LIN {X 0.048,Y -476.705,Z 798.727,A 0.000,B 0.000,C 90.000,E1 346.825} C_DIS
LIN {X -0.156,Y -479.692,Z 798.725,A 0.000,B 0.000,C 90.000,E1 346.589} C_DIS
LIN {X 0.040,Y -487.242,Z 798.722,A 0.000,B 0.000,C 90.000,E1 345.992} C_DIS
LIN {X -0.210,Y -497.903,Z 798.718,A 0.000,B 0.000,C 90.000,E1 345.283} C_DIS
LIN {X -0.076,Y -513.435,Z 798.712,A 0.000,B 0.000,C 90.000,E1 344.212} C_DIS
LIN {X -0.131,Y -527.592,Z 798.707,A 0.000,B 0.000,C 90.000,E1 343.268} C_DIS
LIN {X 0.119,Y -536.840,Z 798.703,A 0.000,B 0.000,C 90.000,E1 342.598} C_DIS
LIN {X 0.066,Y -545.875,Z 798.700,A 0.000,B 0.000,C 90.000,E1 341.945} C_DIS
LIN {X -0.103,Y -553.277,Z 798.697,A 0.000,B 0.000,C 90.000,E1 341.402} C_DIS
LIN {X 0.117,Y -561.468,Z 798.693,A 0.000,B 0.000,C 90.000,E1 340.678} C_DIS
LIN {X 0.102,Y -566.684,Z 798.690,A 0.000,B 0.000,C 90.000,E1 340.188} C_DIS
LIN {X -0.162,Y -570.455,Z 798.688,A 0.000,B 0.000,C 90.000,E1 339.826} C_DIS
LIN {X 0.032,Y -575.308,Z 798.685,A 0.000,B 0.000,C 90.000,E1 339.263} C_DIS
LIN {X -0.045,Y -580.753,Z 798.681,A 0.000,B 0.000,C 90.000,E1 338.592} C_DIS
LIN {X -0.081,Y -585.828,Z 798.677,A 0.000,B 0.000,C 90.000,E1 337.922} C_DIS
LIN {X 0.150,Y -590.581,Z 798.674,A 0.000,B 0.000,C 90.000,E1 337.230} C_DIS
LIN {X -0.352,Y -595.110,Z 798.670,A 0.000,B 0.000,C 90.000,E1 336.613} C_DIS
LIN {X -0.151,Y -601.960,Z 798.664,A 0.000,B 0.000,C 90.000,E1 335.537} C_DIS
LIN {X 0.153,Y -608.398,Z 798.658,A 0.000,B 0.000,C 90.000,E1 334.460} C_DIS
LIN {X 0.000,Y -614.526,Z 798.652,A 0.000,B 0.000,C 90.000,E1 333.435} C_DIS
LIN {X -0.063,Y -618.848,Z 798.648,A 0.000,B 0.000,C 90.000,E1 332.666} C_DIS
LIN {X -0.084,Y -623.726,Z 798.643,A 0.000,B 0.000,C 90.000,E1 331.769} C_DIS
LIN {X -0.071,Y -627.030,Z 798.640,A 0.000,B 0.000,C 90.000,E1 331.129} C_DIS
LIN {X -0.208,Y -633.548,Z 798.633,A 0.000,B 0.000,C 90.000,E1 329.871} C_DIS
LIN {X -0.288,Y -638.306,Z 798.627,A 0.000,B 0.000,C 90.000,E1 328.869} C_DIS
LIN {X 0.182,Y -641.636,Z 798.623,A 0.000,B 0.000,C 90.000,E1 328.074} C_DIS
LIN {X -0.345,Y -645.875,Z 798.617,A 0.000,B 0.000,C 90.000,E1 327.120} C_DIS
LIN {X 0.079,Y -649.887,Z 798.612,A 0.000,B 0.000,C 90.000,E1 326.087} C_DIS
LIN {X 0.096,Y -654.439,Z 798.605,A 0.000,B 0.000,C 90.000,E1 324.848} C_DIS
LIN {X 0.095,Y -657.747,Z 798.599,A 0.000,B 0.000,C 90.000,E1 323.863} C_DIS
LIN {X 0.056,Y -660.091,Z 798.595,A 0.000,B 0.000,C 90.000,E1 323.130} C_DIS
LIN {X 0.062,Y -664.567,Z 798.587,A 0.000,B 0.000,C 90.000,E1 321.662} C_DIS
LIN {X 0.166,Y -667.889,Z 798.580,A 0.000,B 0.000,C 90.000,E1 320.436} C_DIS
LIN {X 0.233,Y -670.845,Z 798.574,A 0.000,B 0.000,C 90.000,E1 319.218} C_DIS
LIN {X -0.082,Y -674.221,Z 798.566,A 0.000,B 0.000,C 90.000,E1 317.796} C_DIS
LIN {X -0.039,Y -675.220,Z 798.563,A 0.000,B 0.000,C 90.000,E1 317.310} C_DIS
LIN {X -0.389,Y -677.131,Z 798.557,A 0.000,B 0.000,C 90.000,E1 316.377} C_DIS
LIN {X -0.248,Y -678.801,Z 798.552,A 0.000,B 0.000,C 90.000,E1 315.405} C_DIS
LIN {X -0.037,Y -680.720,Z 798.546,A 0.000,B 0.000,C 90.000,E1 314.190} C_DIS
LIN {X -0.219,Y -682.747,Z 798.538,A 0.000,B 0.000,C 90.000,E1 312.771} C_DIS
LIN {X 0.089,Y -684.304,Z 798.531,A 0.000,B 0.000,C 90.000,E1 311.553} C_DIS
LIN {X -0.147,Y -685.497,Z 798.526,A 0.000,B 0.000,C 90.000,E1 310.620} C_DIS
LIN {X 0.198,Y -686.778,Z 798.519,A 0.000,B 0.000,C 90.000,E1 309.402} C_DIS
LIN {X 0.120,Y -687.963,Z 798.512,A 0.000,B 0.000,C 90.000,E1 308.222} C_DIS
LIN {X 0.232,Y -689.299,Z 798.505,A 0.000,B 0.000,C 90.000,E1 306.790} C_DIS
LIN {X -0.032,Y -690.506,Z 798.497,A 0.000,B 0.000,C 90.000,E1 305.391} C_DIS
LIN {X 0.090,Y -691.413,Z 798.490,A 0.000,B 0.000,C 90.000,E1 304.199} C_DIS
LIN {X 0.084,Y -692.648,Z 798.481,A 0.000,B 0.000,C 90.000,E1 302.546} C_DIS
LIN {X -0.033,Y -694.068,Z 798.470,A 0.000,B 0.000,C 90.000,E1 300.669} C_DIS
LIN {X -0.004,Y -694.849,Z 798.464,A 0.000,B 0.000,C 90.000,E1 299.489} C_DIS
LIN {X -0.063,Y -695.800,Z 798.455,A 0.000,B 0.000,C 90.000,E1 297.847} C_DIS
LIN {X -0.177,Y -696.974,Z 798.444,A 0.000,B 0.000,C 90.000,E1 295.976} C_DIS
LIN {X 0.197,Y -697.824,Z 798.438,A 0.000,B 0.000,C 90.000,E1 294.771} C_DIS
LIN {X -0.204,Y -697.968,Z 798.435,A 0.000,B 0.000,C 90.000,E1 294.335} C_DIS
LIN {X 0.058,Y -697.877,Z 798.434,A 0.000,B 0.000,C 90.000,E1 294.079} C_DIS
LIN {X -0.342,Y -697.307,Z 798.431,A 0.000,B 0.000,C 90.000,E1 293.643} C_DIS
LIN {X -0.083,Y -696.495,Z 798.430,A 0.000,B 0.000,C 90.000,E1 293.387} C_DIS
LIN {X 0.150,Y -693.935,Z 798.427,A 0.000,B 0.000,C 90.000,E1 292.898} C_DIS
LIN {X 0.272,Y -693.079,Z 798.427,A 0.000,B 0.000,C 90.000,E1 292.770} C_DIS
LIN {X 0.394,Y -691.818,Z 798.426,A 0.000,B 0.000,C 90.000,E1 292.642} C_DIS
LIN {X -0.180,Y -687.922,Z 798.425,A 0.000,B 0.000,C 90.000,E1 292.461} C_DIS
LIN {X -0.053,Y -684.888,Z 798.424,A 0.000,B 0.000,C 90.000,E1 292.280} C_DIS
LIN {X -0.186,Y -683.041,Z 798.423,A 0.000,B 0.000,C 90.000,E1 292.206} C_DIS
LIN {X -0.099,Y -674.904,Z 798.422,A 0.000,B 0.000,C 90.000,E1 291.950} C_DIS
LIN {X -0.081,Y -673.076,Z 798.422,A 0.000,B 0.000,C 90.000,E1 291.897} C_DIS
LIN {X 0.152,Y -663.499,Z 798.421,A 0.000,B 0.000,C 90.000,E1 291.716} C_DIS
LIN {X -0.331,Y -649.518,Z 798.420,A 0.000,B 0.000,C 90.000,E1 291.535} C_DIS
LIN {X -0.273,Y -635.379,Z 798.418,A 0.000,B 0.000,C 90.000,E1 291.280} C_DIS
LIN {X -0.207,Y -618.231,Z 798.416,A 0.000,B 0.000,C 90.000,E1 290.918} C_DIS
LIN {X 0.086,Y -605.022,Z 798.414,A 0.000,B 0.000,C 90.000,E1 290.556} C_DIS
LIN {X -0.042,Y -598.409,Z 798.413,A 0.000,B 0.000,C 90.000,E1 290.375} C_DIS
LIN {X -0.004,Y -585.106,Z 798.411,A 0.000,B 0.000,C 90.000,E1 289.939} C_DIS
LIN {X 0.004,Y -574.115,Z 798.408,A 0.000,B 0.000,C 90.000,E1 289.504} C_DIS
LIN {X -0.070,Y -568.690,Z 798.407,A 0.000,B 0.000,C 90.000,E1 289.214} C_DIS
LIN {X -0.174,Y -566.213,Z 798.405,A 0.000,B 0.000,C 90.000,E1 288.960} C_DIS
LIN {X -0.111,Y -565.126,Z 798.405,A 0.000,B 0.000,C 90.000,E1 288.852} C_DIS
LIN {X -0.016,Y -564.192,Z 798.404,A 0.000,B 0.000,C 90.000,E1 288.671} C_DIS
LIN {X -0.119,Y -563.612,Z 798.403,A 0.000,B 0.000,C 90.000,E1 288.544} C_DIS
LIN {X 0.123,Y -563.320,Z 798.402,A 0.000,B 0.000,C 90.000,E1 288.362} C_DIS
LIN {X -0.095,Y -562.507,Z 798.401,A 0.000,B 0.000,C 90.000,E1 288.109} C_DIS
LIN {X 0.045,Y -562.296,Z 798.399,A 0.000,B 0.000,C 90.000,E1 287.819} C_DIS
LIN {X 0.186,Y -562.165,Z 798.398,A 0.000,B 0.000,C 90.000,E1 287.528} C_DIS
LIN {X 0.073,Y -562.226,Z 798.397,A 0.000,B 0.000,C 90.000,E1 287.402} C_DIS
LIN {X -0.127,Y -564.221,Z 798.393,A 0.000,B 0.000,C 90.000,E1 286.732} C_DIS
LIN {X 0.136,Y -565.076,Z 798.392,A 0.000,B 0.000,C 90.000,E1 286.567} C_DIS
LIN {X 0.180,Y -568.381,Z 798.390,A 0.000,B 0.000,C 90.000,E1 286.150} C_DIS
LIN {X 0.070,Y -569.256,Z 798.389,A 0.000,B 0.000,C 90.000,E1 286.024} C_DIS
LIN {X -0.235,Y -572.706,Z 798.385,A 0.000,B 0.000,C 90.000,E1 285.371} C_DIS
LIN {X 0.103,Y -573.656,Z 798.384,A 0.000,B 0.000,C 90.000,E1 285.064} C_DIS
LIN {X -0.220,Y -576.381,Z 798.378,A 0.000,B 0.000,C 90.000,E1 284.008} C_DIS
LIN {X -0.013,Y -576.591,Z 798.376,A 0.000,B 0.000,C 90.000,E1 283.716} C_DIS
LIN {X -0.020,Y -576.495,Z 798.373,A 0.000,B 0.000,C 90.000,E1 283.175} C_DIS
LIN {X 0.190,Y -576.235,Z 798.372,A 0.000,B 0.000,C 90.000,E1 282.883} C_DIS
LIN {X -0.161,Y -575.837,Z 798.370,A 0.000,B 0.000,C 90.000,E1 282.647} C_DIS
LIN {X 0.256,Y -573.735,Z 798.367,A 0.000,B 0.000,C 90.000,E1 282.063} C_DIS
LIN {X -0.100,Y -572.413,Z 798.366,A 0.000,B 0.000,C 90.000,E1 281.827} C_DIS
LIN {X -0.143,Y -569.026,Z 798.363,A 0.000,B 0.000,C 90.000,E1 281.422} C_DIS
LIN {X 0.123,Y -566.344,Z 798.362,A 0.000,B 0.000,C 90.000,E1 281.130} C_DIS
LIN {X 0.232,Y -562.560,Z 798.361,A 0.000,B 0.000,C 90.000,E1 280.894} C_DIS
LIN {X -0.156,Y -560.238,Z 798.360,A 0.000,B 0.000,C 90.000,E1 280.838} C_DIS
LIN {X -0.294,Y -558.014,Z 798.360,A 0.000,B 0.000,C 90.000,E1 280.782} C_DIS
LIN {X 0.219,Y -556.305,Z 798.359,A 0.000,B 0.000,C 90.000,E1 280.658} C_DIS
LIN {X -0.099,Y -555.281,Z 798.359,A 0.000,B 0.000,C 90.000,E1 280.602} C_DIS
LIN {X -0.134,Y -552.696,Z 798.357,A 0.000,B 0.000,C 90.000,E1 280.310} C_DIS
LIN {X 0.133,Y -552.209,Z 798.357,A 0.000,B 0.000,C 90.000,E1 280.197} C_DIS
LIN {X 0.017,Y -551.503,Z 798.354,A 0.000,B 0.000,C 90.000,E1 279.792} C_DIS
LIN {X 0.215,Y -550.863,Z 798.342,A 0.000,B 0.000,C 90.000,E1 277.530} C_DIS
LIN {X 0.166,Y -550.166,Z 798.333,A 0.000,B 0.000,C 90.000,E1 275.853} C_DIS
LIN {X -0.105,Y -549.616,Z 798.326,A 0.000,B 0.000,C 90.000,E1 274.759} C_DIS
LIN {X 0.122,Y -548.967,Z 798.320,A 0.000,B 0.000,C 90.000,E1 273.612} C_DIS
LIN {X -0.108,Y -547.797,Z 798.311,A 0.000,B 0.000,C 90.000,E1 271.949} C_DIS
LIN {X 0.140,Y -546.886,Z 798.303,A 0.000,B 0.000,C 90.000,E1 270.516} C_DIS
LIN {X -0.187,Y -545.959,Z 798.295,A 0.000,B 0.000,C 90.000,E1 269.141} C_DIS
LIN {X 0.097,Y -544.570,Z 798.284,A 0.000,B 0.000,C 90.000,E1 267.135} C_DIS
LIN {X -0.201,Y -543.491,Z 798.275,A 0.000,B 0.000,C 90.000,E1 265.469} C_DIS
LIN {X -0.003,Y -542.620,Z 798.267,A 0.000,B 0.000,C 90.000,E1 264.033} C_DIS
LIN {X 0.229,Y -541.566,Z 798.259,A 0.000,B 0.000,C 90.000,E1 262.591} C_DIS
LIN {X 0.059,Y -540.107,Z 798.250,A 0.000,B 0.000,C 90.000,E1 260.905} C_DIS
LIN {X 0.257,Y -539.053,Z 798.243,A 0.000,B 0.000,C 90.000,E1 259.746} C_DIS
LIN {X 0.139,Y -537.415,Z 798.234,A 0.000,B 0.000,C 90.000,E1 258.049} C_DIS
LIN {X -0.019,Y -535.728,Z 798.224,A 0.000,B 0.000,C 90.000,E1 256.353} C_DIS
LIN {X -0.147,Y -534.186,Z 798.216,A 0.000,B 0.000,C 90.000,E1 254.936} C_DIS
LIN {X 0.022,Y -532.181,Z 798.207,A 0.000,B 0.000,C 90.000,E1 253.196} C_DIS
LIN {X -0.030,Y -530.495,Z 798.199,A 0.000,B 0.000,C 90.000,E1 251.764} C_DIS
LIN {X 0.041,Y -528.664,Z 798.191,A 0.000,B 0.000,C 90.000,E1 250.315} C_DIS
LIN {X 0.078,Y -527.108,Z 798.184,A 0.000,B 0.000,C 90.000,E1 249.156} C_DIS
LIN {X 0.139,Y -524.559,Z 798.175,A 0.000,B 0.000,C 90.000,E1 247.411} C_DIS
LIN {X 0.153,Y -521.953,Z 798.165,A 0.000,B 0.000,C 90.000,E1 245.665} C_DIS
LIN {X 0.178,Y -519.658,Z 798.157,A 0.000,B 0.000,C 90.000,E1 244.204} C_DIS
LIN {X 0.157,Y -517.176,Z 798.149,A 0.000,B 0.000,C 90.000,E1 242.743} C_DIS
LIN {X -0.133,Y -514.636,Z 798.141,A 0.000,B 0.000,C 90.000,E1 241.307} C_DIS
LIN {X 0.230,Y -511.862,Z 798.132,A 0.000,B 0.000,C 90.000,E1 239.793} C_DIS
LIN {X -0.238,Y -509.540,Z 798.126,A 0.000,B 0.000,C 90.000,E1 238.663} C_DIS
LIN {X -0.145,Y -506.520,Z 798.118,A 0.000,B 0.000,C 90.000,E1 237.168} C_DIS
LIN {X -0.004,Y -503.984,Z 798.111,A 0.000,B 0.000,C 90.000,E1 235.960} C_DIS
LIN {X -0.277,Y -499.922,Z 798.101,A 0.000,B 0.000,C 90.000,E1 234.196} C_DIS
LIN {X 0.189,Y -496.161,Z 798.093,A 0.000,B 0.000,C 90.000,E1 232.637} C_DIS
LIN {X -0.042,Y -491.609,Z 798.083,A 0.000,B 0.000,C 90.000,E1 230.848} C_DIS
LIN {X 0.130,Y -485.202,Z 798.067,A 0.000,B 0.000,C 90.000,E1 228.081} C_DIS
LIN {X -0.249,Y -480.588,Z 798.055,A 0.000,B 0.000,C 90.000,E1 225.972} C_DIS
LIN {X -0.195,Y -476.476,Z 798.045,A 0.000,B 0.000,C 90.000,E1 224.109} C_DIS
LIN {X -0.127,Y -471.709,Z 798.033,A 0.000,B 0.000,C 90.000,E1 221.919} C_DIS
LIN {X 0.088,Y -467.690,Z 798.022,A 0.000,B 0.000,C 90.000,E1 220.011} C_DIS
LIN {X -0.146,Y -464.455,Z 798.014,A 0.000,B 0.000,C 90.000,E1 218.463} C_DIS
LIN {X 0.059,Y -459.854,Z 798.001,A 0.000,B 0.000,C 90.000,E1 216.217} C_DIS
LIN {X -0.136,Y -455.828,Z 797.991,A 0.000,B 0.000,C 90.000,E1 214.326} C_DIS
LIN {X 0.038,Y -451.298,Z 797.978,A 0.000,B 0.000,C 90.000,E1 212.054} C_DIS
LIN {X -0.082,Y -447.415,Z 797.967,A 0.000,B 0.000,C 90.000,E1 210.129} C_DIS
LIN {X 0.097,Y -443.579,Z 797.957,A 0.000,B 0.000,C 90.000,E1 208.153} C_DIS
LIN {X -0.070,Y -440.543,Z 797.947,A 0.000,B 0.000,C 90.000,E1 206.539} C_DIS
LIN {X 0.155,Y -436.121,Z 797.935,A 0.000,B 0.000,C 90.000,E1 204.207} C_DIS
LIN {X -0.125,Y -432.889,Z 797.925,A 0.000,B 0.000,C 90.000,E1 202.589} C_DIS
LIN {X -0.067,Y -429.687,Z 797.916,A 0.000,B 0.000,C 90.000,E1 200.918} C_DIS
LIN {X 0.170,Y -425.220,Z 797.903,A 0.000,B 0.000,C 90.000,E1 198.544} C_DIS
LIN {X -0.001,Y -422.607,Z 797.896,A 0.000,B 0.000,C 90.000,E1 197.221} C_DIS
LIN {X -0.160,Y -419.352,Z 797.886,A 0.000,B 0.000,C 90.000,E1 195.552} C_DIS
LIN {X 0.210,Y -414.775,Z 797.873,A 0.000,B 0.000,C 90.000,E1 193.119} C_DIS
LIN {X 0.023,Y -412.875,Z 797.867,A 0.000,B 0.000,C 90.000,E1 192.119} C_DIS
LIN {X -0.075,Y -408.571,Z 797.854,A 0.000,B 0.000,C 90.000,E1 189.726} C_DIS
LIN {X -0.059,Y -406.165,Z 797.846,A 0.000,B 0.000,C 90.000,E1 188.341} C_DIS
LIN {X -0.021,Y -403.637,Z 797.839,A 0.000,B 0.000,C 90.000,E1 186.947} C_DIS
LIN {X -0.135,Y -400.464,Z 797.829,A 0.000,B 0.000,C 90.000,E1 185.220} C_DIS
LIN {X -0.017,Y -393.717,Z 797.804,A 0.000,B 0.000,C 90.000,E1 180.630} C_DIS
LIN {X 0.090,Y -390.124,Z 797.786,A 0.000,B 0.000,C 90.000,E1 177.421} C_DIS
LIN {X -0.025,Y -387.841,Z 797.774,A 0.000,B 0.000,C 90.000,E1 175.298} C_DIS
LIN {X -0.132,Y -385.637,Z 797.762,A 0.000,B 0.000,C 90.000,E1 173.166} C_DIS
LIN {X 0.135,Y -383.530,Z 797.750,A 0.000,B 0.000,C 90.000,E1 170.971} C_DIS
LIN {X -0.083,Y -381.070,Z 797.734,A 0.000,B 0.000,C 90.000,E1 168.117} C_DIS
LIN {X -0.140,Y -378.783,Z 797.716,A 0.000,B 0.000,C 90.000,E1 164.866} C_DIS
LIN {X -0.097,Y -376.970,Z 797.694,A 0.000,B 0.000,C 90.000,E1 160.859} C_DIS
LIN {X 0.037,Y -377.905,Z 797.649,A 0.000,B 0.000,C 90.000,E1 152.820} C_DIS
LIN {X 0.180,Y -380.213,Z 797.635,A 0.000,B 0.000,C 90.000,E1 150.255} C_DIS
LIN {X -0.052,Y -381.817,Z 797.629,A 0.000,B 0.000,C 90.000,E1 149.203} C_DIS
LIN {X 0.077,Y -384.673,Z 797.621,A 0.000,B 0.000,C 90.000,E1 147.740} C_DIS
LIN {X 0.136,Y -388.637,Z 797.613,A 0.000,B 0.000,C 90.000,E1 146.294} C_DIS
LIN {X -0.125,Y -392.389,Z 797.607,A 0.000,B 0.000,C 90.000,E1 145.261} C_DIS
LIN {X 0.107,Y -394.977,Z 797.604,A 0.000,B 0.000,C 90.000,E1 144.609} C_DIS
LIN {X 0.058,Y -398.597,Z 797.600,A 0.000,B 0.000,C 90.000,E1 143.909} C_DIS
LIN {X 0.009,Y -402.309,Z 797.596,A 0.000,B 0.000,C 90.000,E1 143.290} C_DIS
LIN {X 0.188,Y -407.473,Z 797.592,A 0.000,B 0.000,C 90.000,E1 142.477} C_DIS
LIN {X 0.122,Y -416.188,Z 797.585,A 0.000,B 0.000,C 90.000,E1 141.331} C_DIS
LIN {X -0.063,Y -425.883,Z 797.579,A 0.000,B 0.000,C 90.000,E1 140.194} C_DIS
LIN {X 0.075,Y -433.645,Z 797.573,A 0.000,B 0.000,C 90.000,E1 139.175} C_DIS
LIN {X 0.162,Y -446.410,Z 797.564,A 0.000,B 0.000,C 90.000,E1 137.553} C_DIS
LIN {X 0.166,Y -451.691,Z 797.561,A 0.000,B 0.000,C 90.000,E1 136.905} C_DIS
LIN {X 0.078,Y -459.089,Z 797.555,A 0.000,B 0.000,C 90.000,E1 135.972} C_DIS
LIN {X -0.001,Y -463.712,Z 797.552,A 0.000,B 0.000,C 90.000,E1 135.364} C_DIS
LIN {X 0.007,Y -473.709,Z 797.544,A 0.000,B 0.000,C 90.000,E1 133.947} C_DIS
LIN {X 0.141,Y -480.131,Z 797.539,A 0.000,B 0.000,C 90.000,E1 133.014} C_DIS
LIN {X 0.268,Y -487.242,Z 797.533,A 0.000,B 0.000,C 90.000,E1 131.919} C_DIS
LIN {X 0.248,Y -495.005,Z 797.526,A 0.000,B 0.000,C 90.000,E1 130.701} C_DIS
LIN {X 0.117,Y -502.992,Z 797.519,A 0.000,B 0.000,C 90.000,E1 129.358} C_DIS
LIN {X -0.004,Y -507.287,Z 797.515,A 0.000,B 0.000,C 90.000,E1 128.624} C_DIS
LIN {X -0.059,Y -513.696,Z 797.508,A 0.000,B 0.000,C 90.000,E1 127.443} C_DIS
LIN {X -0.279,Y -518.187,Z 797.503,A 0.000,B 0.000,C 90.000,E1 126.583} C_DIS
LIN {X -0.028,Y -522.549,Z 797.498,A 0.000,B 0.000,C 90.000,E1 125.678} C_DIS
LIN {X -0.024,Y -527.143,Z 797.493,A 0.000,B 0.000,C 90.000,E1 124.692} C_DIS
LIN {X 0.002,Y -533.141,Z 797.485,A 0.000,B 0.000,C 90.000,E1 123.245} C_DIS
LIN {X -0.322,Y -536.545,Z 797.480,A 0.000,B 0.000,C 90.000,E1 122.418} C_DIS
LIN {X -0.157,Y -540.829,Z 797.474,A 0.000,B 0.000,C 90.000,E1 121.258} C_DIS
LIN {X 0.051,Y -543.851,Z 797.469,A 0.000,B 0.000,C 90.000,E1 120.384} C_DIS
LIN {X -0.232,Y -547.520,Z 797.463,A 0.000,B 0.000,C 90.000,E1 119.283} C_DIS
LIN {X 0.055,Y -551.711,Z 797.455,A 0.000,B 0.000,C 90.000,E1 117.847} C_DIS
LIN {X -0.152,Y -553.269,Z 797.452,A 0.000,B 0.000,C 90.000,E1 117.308} C_DIS
LIN {X 0.163,Y -555.267,Z 797.447,A 0.000,B 0.000,C 90.000,E1 116.437} C_DIS
LIN {X 0.039,Y -557.302,Z 797.441,A 0.000,B 0.000,C 90.000,E1 115.335} C_DIS
LIN {X 0.118,Y -558.260,Z 797.438,A 0.000,B 0.000,C 90.000,E1 114.771} C_DIS
LIN {X -0.213,Y -559.661,Z 797.432,A 0.000,B 0.000,C 90.000,E1 113.695} C_DIS
LIN {X -0.235,Y -560.865,Z 797.425,A 0.000,B 0.000,C 90.000,E1 112.589} C_DIS
LIN {X 0.088,Y -562.248,Z 797.418,A 0.000,B 0.000,C 90.000,E1 111.173} C_DIS
LIN {X -0.097,Y -563.346,Z 797.410,A 0.000,B 0.000,C 90.000,E1 109.812} C_DIS
LIN {X 0.065,Y -564.073,Z 797.402,A 0.000,B 0.000,C 90.000,E1 108.417} C_DIS
LIN {X -0.321,Y -564.895,Z 797.393,A 0.000,B 0.000,C 90.000,E1 106.804} C_DIS
LIN {X 0.170,Y -565.967,Z 797.383,A 0.000,B 0.000,C 90.000,E1 104.828} C_DIS
LIN {X -0.161,Y -567.198,Z 797.372,A 0.000,B 0.000,C 90.000,E1 102.939} C_DIS
LIN {X 0.164,Y -568.222,Z 797.364,A 0.000,B 0.000,C 90.000,E1 101.535} C_DIS
LIN {X -0.156,Y -569.282,Z 797.357,A 0.000,B 0.000,C 90.000,E1 100.197} C_DIS
LIN {X 0.109,Y -570.390,Z 797.349,A 0.000,B 0.000,C 90.000,E1 98.803} C_DIS
LIN {X -0.069,Y -571.516,Z 797.340,A 0.000,B 0.000,C 90.000,E1 97.182} C_DIS
LIN {X -0.034,Y -572.182,Z 797.334,A 0.000,B 0.000,C 90.000,E1 96.087} C_DIS
LIN {X -0.115,Y -573.264,Z 797.323,A 0.000,B 0.000,C 90.000,E1 94.188} C_DIS
LIN {X -0.067,Y -573.781,Z 797.317,A 0.000,B 0.000,C 90.000,E1 93.094} C_DIS
LIN {X 0.235,Y -574.510,Z 797.308,A 0.000,B 0.000,C 90.000,E1 91.432} C_DIS
LIN {X -0.180,Y -574.948,Z 797.301,A 0.000,B 0.000,C 90.000,E1 90.115} C_DIS
LIN {X 0.139,Y -575.545,Z 797.292,A 0.000,B 0.000,C 90.000,E1 88.453} C_DIS
LIN {X -0.068,Y -575.967,Z 797.282,A 0.000,B 0.000,C 90.000,E1 86.846} C_DIS
LIN {X -0.107,Y -576.439,Z 797.272,A 0.000,B 0.000,C 90.000,E1 84.951} C_DIS
LIN {X 0.136,Y -576.695,Z 797.264,A 0.000,B 0.000,C 90.000,E1 83.571} C_DIS
LIN {X 0.079,Y -576.993,Z 797.255,A 0.000,B 0.000,C 90.000,E1 81.951} C_DIS
LIN {X 0.029,Y -577.292,Z 797.246,A 0.000,B 0.000,C 90.000,E1 80.330} C_DIS
LIN {X -0.141,Y -577.537,Z 797.239,A 0.000,B 0.000,C 90.000,E1 78.993} C_DIS
LIN {X -0.197,Y -577.585,Z 797.231,A 0.000,B 0.000,C 90.000,E1 77.645} C_DIS
LIN {X 0.099,Y -577.526,Z 797.222,A 0.000,B 0.000,C 90.000,E1 75.992} C_DIS
LIN {X 0.184,Y -577.316,Z 797.215,A 0.000,B 0.000,C 90.000,E1 74.629} C_DIS
LIN {X 0.073,Y -577.068,Z 797.206,A 0.000,B 0.000,C 90.000,E1 73.015} C_DIS
LIN {X 0.306,Y -576.761,Z 797.198,A 0.000,B 0.000,C 90.000,E1 71.638} C_DIS
LIN {X -0.207,Y -576.390,Z 797.192,A 0.000,B 0.000,C 90.000,E1 70.604} C_DIS
LIN {X 0.189,Y -575.896,Z 797.185,A 0.000,B 0.000,C 90.000,E1 69.209} C_DIS
LIN {X -0.133,Y -575.419,Z 797.179,A 0.000,B 0.000,C 90.000,E1 68.156} C_DIS
LIN {X -0.088,Y -574.714,Z 797.171,A 0.000,B 0.000,C 90.000,E1 66.794} C_DIS
LIN {X 0.331,Y -574.047,Z 797.165,A 0.000,B 0.000,C 90.000,E1 65.665} C_DIS
LIN {X 0.218,Y -573.334,Z 797.159,A 0.000,B 0.000,C 90.000,E1 64.588} C_DIS
LIN {X 0.095,Y -572.520,Z 797.153,A 0.000,B 0.000,C 90.000,E1 63.512} C_DIS
LIN {X 0.216,Y -571.490,Z 797.147,A 0.000,B 0.000,C 90.000,E1 62.410} C_DIS
LIN {X -0.283,Y -570.602,Z 797.142,A 0.000,B 0.000,C 90.000,E1 61.641} C_DIS
LIN {X -0.194,Y -569.232,Z 797.136,A 0.000,B 0.000,C 90.000,E1 60.539} C_DIS
LIN {X 0.152,Y -567.652,Z 797.130,A 0.000,B 0.000,C 90.000,E1 59.410} C_DIS
LIN {X -0.114,Y -566.325,Z 797.126,A 0.000,B 0.000,C 90.000,E1 58.614} C_DIS
LIN {X -0.097,Y -564.856,Z 797.121,A 0.000,B 0.000,C 90.000,E1 57.788} C_DIS
LIN {X -0.089,Y -563.185,Z 797.116,A 0.000,B 0.000,C 90.000,E1 56.962} C_DIS
LIN {X -0.313,Y -560.700,Z 797.110,A 0.000,B 0.000,C 90.000,E1 55.881} C_DIS
LIN {X -0.264,Y -557.786,Z 797.104,A 0.000,B 0.000,C 90.000,E1 54.769} C_DIS
LIN {X -0.011,Y -555.414,Z 797.100,A 0.000,B 0.000,C 90.000,E1 53.909} C_DIS
LIN {X 0.145,Y -553.662,Z 797.096,A 0.000,B 0.000,C 90.000,E1 53.336} C_DIS
LIN {X 0.353,Y -550.803,Z 797.092,A 0.000,B 0.000,C 90.000,E1 52.477} C_DIS
LIN {X -0.298,Y -548.790,Z 797.089,A 0.000,B 0.000,C 90.000,E1 51.984} C_DIS
LIN {X 0.193,Y -545.353,Z 797.084,A 0.000,B 0.000,C 90.000,E1 51.090} C_DIS
LIN {X -0.149,Y -542.914,Z 797.081,A 0.000,B 0.000,C 90.000,E1 50.561} C_DIS
LIN {X -0.094,Y -540.266,Z 797.078,A 0.000,B 0.000,C 90.000,E1 49.989} C_DIS
LIN {X -0.291,Y -534.898,Z 797.072,A 0.000,B 0.000,C 90.000,E1 49.013} C_DIS
LIN {X 0.057,Y -533.336,Z 797.071,A 0.000,B 0.000,C 90.000,E1 48.690} C_DIS
LIN {X -0.200,Y -528.678,Z 797.067,A 0.000,B 0.000,C 90.000,E1 48.000} C_DIS
LIN {X 0.089,Y -524.643,Z 797.063,A 0.000,B 0.000,C 90.000,E1 47.391} C_DIS
LIN {X -0.189,Y -521.357,Z 797.061,A 0.000,B 0.000,C 90.000,E1 46.986} C_DIS
LIN {X 0.040,Y -516.511,Z 797.058,A 0.000,B 0.000,C 90.000,E1 46.377} C_DIS
LIN {X 0.111,Y -507.647,Z 797.052,A 0.000,B 0.000,C 90.000,E1 45.405} C_DIS
LIN {X -0.261,Y -500.374,Z 797.049,A 0.000,B 0.000,C 90.000,E1 44.757} C_DIS
LIN {X -0.219,Y -495.926,Z 797.046,A 0.000,B 0.000,C 90.000,E1 44.352} C_DIS
LIN {X 0.293,Y -489.920,Z 797.044,A 0.000,B 0.000,C 90.000,E1 43.785} C_DIS
LIN {X -0.062,Y -482.139,Z 797.040,A 0.000,B 0.000,C 90.000,E1 43.218} C_DIS
LIN {X 0.189,Y -474.147,Z 797.037,A 0.000,B 0.000,C 90.000,E1 42.609} C_DIS
LIN {X -0.018,Y -464.550,Z 797.033,A 0.000,B 0.000,C 90.000,E1 41.962} C_DIS
LIN {X -0.073,Y -446.893,Z 797.026,A 0.000,B 0.000,C 90.000,E1 40.744} C_DIS
LIN {X -0.233,Y -421.708,Z 797.016,A 0.000,B 0.000,C 90.000,E1 38.910} C_DIS
LIN {X 0.056,Y -407.950,Z 797.010,A 0.000,B 0.000,C 90.000,E1 37.729} C_DIS
LIN {X 0.071,Y -403.546,Z 797.007,A 0.000,B 0.000,C 90.000,E1 37.282} C_DIS
LIN {X 0.028,Y -403.146,Z 797.007,A 0.000,B 0.000,C 90.000,E1 37.237} C_DIS
LIN {X -0.001,Y -403.124,Z 797.007,A 0.000,B 0.000,C 90.000,E1 37.237} C_DIS
LIN {X 0.126,Y -395.009,Z 796.982,A 0.000,B 0.000,C 90.000,E1 32.673} C_DIS
LIN {X -0.212,Y -394.922,Z 796.981,A 0.000,B 0.000,C 90.000,E1 32.546} C_DIS
LIN {X -0.152,Y -395.864,Z 796.966,A 0.000,B 0.000,C 90.000,E1 29.873} C_DIS
LIN {X 0.205,Y -397.336,Z 796.950,A 0.000,B 0.000,C 90.000,E1 27.001} C_DIS
LIN {X 0.140,Y -398.604,Z 796.938,A 0.000,B 0.000,C 90.000,E1 24.899} C_DIS
LIN {X -0.053,Y -400.889,Z 796.921,A 0.000,B 0.000,C 90.000,E1 21.770} C_DIS
LIN {X 0.236,Y -404.220,Z 796.902,A 0.000,B 0.000,C 90.000,E1 18.236} C_DIS
LIN {X -0.208,Y -409.195,Z 796.880,A 0.000,B 0.000,C 90.000,E1 14.481} C_DIS
LIN {X -0.128,Y -413.616,Z 796.865,A 0.000,B 0.000,C 90.000,E1 11.715} C_DIS
LIN {X -0.189,Y -417.166,Z 796.854,A 0.000,B 0.000,C 90.000,E1 9.670} C_DIS
LIN {X 0.044,Y -420.183,Z 796.844,A 0.000,B 0.000,C 90.000,E1 7.936} C_DIS
LIN {X -0.001,Y -423.832,Z 796.833,A 0.000,B 0.000,C 90.000,E1 5.910} C_DIS
LIN {X -0.056,Y -427.559,Z 796.822,A 0.000,B 0.000,C 90.000,E1 3.898} C_DIS
LIN {X -0.069,Y -431.408,Z 796.810,A 0.000,B 0.000,C 90.000,E1 1.892} C_DIS
LIN {X 0.165,Y -435.686,Z 796.799,A 0.000,B 0.000,C 90.000,E1 359.771} C_DIS
LIN {X 0.142,Y -441.483,Z 796.784,A 0.000,B 0.000,C 90.000,E1 357.135} C_DIS
LIN {X 0.208,Y -446.922,Z 796.771,A 0.000,B 0.000,C 90.000,E1 354.837} C_DIS
LIN {X 0.130,Y -450.859,Z 796.763,A 0.000,B 0.000,C 90.000,E1 353.223} C_DIS
LIN {X 0.186,Y -454.754,Z 796.754,A 0.000,B 0.000,C 90.000,E1 351.602} C_DIS
LIN {X -0.126,Y -460.338,Z 796.741,A 0.000,B 0.000,C 90.000,E1 349.398} C_DIS
LIN {X 0.065,Y -462.950,Z 796.737,A 0.000,B 0.000,C 90.000,E1 348.578} C_DIS
LIN {X -0.142,Y -464.261,Z 796.735,A 0.000,B 0.000,C 90.000,E1 348.285} C_DIS
LIN {X 0.112,Y -465.806,Z 796.733,A 0.000,B 0.000,C 90.000,E1 347.937} C_DIS
LIN {X -0.045,Y -468.262,Z 796.731,A 0.000,B 0.000,C 90.000,E1 347.589} C_DIS
LIN {X 0.002,Y -473.215,Z 796.728,A 0.000,B 0.000,C 90.000,E1 346.992} C_DIS
LIN {X -0.049,Y -481.413,Z 796.724,A 0.000,B 0.000,C 90.000,E1 346.284} C_DIS
LIN {X 0.163,Y -490.454,Z 796.720,A 0.000,B 0.000,C 90.000,E1 345.589} C_DIS
LIN {X -0.228,Y -509.270,Z 796.713,A 0.000,B 0.000,C 90.000,E1 344.338} C_DIS
LIN {X 0.045,Y -526.667,Z 796.706,A 0.000,B 0.000,C 90.000,E1 343.142} C_DIS
LIN {X 0.198,Y -535.950,Z 796.703,A 0.000,B 0.000,C 90.000,E1 342.489} C_DIS
LIN {X -0.208,Y -546.506,Z 796.699,A 0.000,B 0.000,C 90.000,E1 341.764} C_DIS
LIN {X 0.242,Y -552.410,Z 796.696,A 0.000,B 0.000,C 90.000,E1 341.275} C_DIS
LIN {X -0.079,Y -560.796,Z 796.692,A 0.000,B 0.000,C 90.000,E1 340.604} C_DIS
LIN {X -0.156,Y -566.114,Z 796.690,A 0.000,B 0.000,C 90.000,E1 340.115} C_DIS
LIN {X 0.061,Y -571.128,Z 796.687,A 0.000,B 0.000,C 90.000,E1 339.571} C_DIS
LIN {X 0.107,Y -575.854,Z 796.684,A 0.000,B 0.000,C 90.000,E1 339.028} C_DIS
LIN {X -0.044,Y -582.271,Z 796.679,A 0.000,B 0.000,C 90.000,E1 338.230} C_DIS
LIN {X 0.090,Y -588.207,Z 796.675,A 0.000,B 0.000,C 90.000,E1 337.411} C_DIS
LIN {X 0.013,Y -594.698,Z 796.669,A 0.000,B 0.000,C 90.000,E1 336.485} C_DIS
LIN {X 0.214,Y -601.571,Z 796.664,A 0.000,B 0.000,C 90.000,E1 335.409} C_DIS
LIN {X -0.294,Y -608.046,Z 796.658,A 0.000,B 0.000,C 90.000,E1 334.409} C_DIS
LIN {X 0.071,Y -614.941,Z 796.651,A 0.000,B 0.000,C 90.000,E1 333.204} C_DIS
LIN {X 0.015,Y -618.553,Z 796.648,A 0.000,B 0.000,C 90.000,E1 332.564} C_DIS
LIN {X 0.277,Y -624.182,Z 796.642,A 0.000,B 0.000,C 90.000,E1 331.513} C_DIS
LIN {X 0.088,Y -630.106,Z 796.636,A 0.000,B 0.000,C 90.000,E1 330.383} C_DIS
LIN {X 0.151,Y -633.403,Z 796.632,A 0.000,B 0.000,C 90.000,E1 329.744} C_DIS
LIN {X 0.092,Y -638.739,Z 796.626,A 0.000,B 0.000,C 90.000,E1 328.614} C_DIS
LIN {X 0.070,Y -643.127,Z 796.620,A 0.000,B 0.000,C 90.000,E1 327.612} C_DIS
LIN {X 0.393,Y -646.307,Z 796.616,A 0.000,B 0.000,C 90.000,E1 326.834} C_DIS
LIN {X -0.139,Y -649.326,Z 796.612,A 0.000,B 0.000,C 90.000,E1 326.135} C_DIS
LIN {X -0.125,Y -653.966,Z 796.605,A 0.000,B 0.000,C 90.000,E1 324.895} C_DIS
LIN {X -0.125,Y -657.346,Z 796.599,A 0.000,B 0.000,C 90.000,E1 323.909} C_DIS
LIN {X 0.363,Y -659.724,Z 796.595,A 0.000,B 0.000,C 90.000,E1 323.130} C_DIS
LIN {X 0.394,Y -663.496,Z 796.589,A 0.000,B 0.000,C 90.000,E1 321.904} C_DIS
LIN {X 0.419,Y -665.599,Z 796.585,A 0.000,B 0.000,C 90.000,E1 321.170} C_DIS
LIN {X -0.049,Y -667.649,Z 796.580,A 0.000,B 0.000,C 90.000,E1 320.481} C_DIS
LIN {X 0.091,Y -670.689,Z 796.574,A 0.000,B 0.000,C 90.000,E1 319.256} C_DIS
LIN {X -0.304,Y -673.576,Z 796.567,A 0.000,B 0.000,C 90.000,E1 318.081} C_DIS
LIN {X 0.234,Y -674.718,Z 796.564,A 0.000,B 0.000,C 90.000,E1 317.553} C_DIS
LIN {X -0.093,Y -677.132,Z 796.558,A 0.000,B 0.000,C 90.000,E1 316.377} C_DIS
LIN {X 0.049,Y -678.799,Z 796.552,A 0.000,B 0.000,C 90.000,E1 315.405} C_DIS
LIN {X 0.261,Y -680.787,Z 796.546,A 0.000,B 0.000,C 90.000,E1 314.190} C_DIS
LIN {X 0.082,Y -682.855,Z 796.538,A 0.000,B 0.000,C 90.000,E1 312.771} C_DIS
LIN {X -0.120,Y -684.435,Z 796.531,A 0.000,B 0.000,C 90.000,E1 311.595} C_DIS
LIN {X 0.104,Y -685.376,Z 796.527,A 0.000,B 0.000,C 90.000,E1 310.862} C_DIS
LIN {X -0.075,Y -686.693,Z 796.521,A 0.000,B 0.000,C 90.000,E1 309.688} C_DIS
LIN {X 0.005,Y -688.135,Z 796.513,A 0.000,B 0.000,C 90.000,E1 308.257} C_DIS
LIN {X -0.418,Y -689.476,Z 796.505,A 0.000,B 0.000,C 90.000,E1 306.870} C_DIS
LIN {X 0.088,Y -690.524,Z 796.498,A 0.000,B 0.000,C 90.000,E1 305.644} C_DIS
LIN {X -0.190,Y -691.431,Z 796.492,A 0.000,B 0.000,C 90.000,E1 304.485} C_DIS
LIN {X 0.411,Y -692.849,Z 796.481,A 0.000,B 0.000,C 90.000,E1 302.546} C_DIS
LIN {X -0.055,Y -694.450,Z 796.469,A 0.000,B 0.000,C 90.000,E1 300.463} C_DIS
LIN {X -0.023,Y -695.181,Z 796.463,A 0.000,B 0.000,C 90.000,E1 299.283} C_DIS
LIN {X -0.082,Y -696.112,Z 796.454,A 0.000,B 0.000,C 90.000,E1 297.641} C_DIS
LIN {X -0.199,Y -697.264,Z 796.443,A 0.000,B 0.000,C 90.000,E1 295.771} C_DIS
LIN {X -0.088,Y -697.928,Z 796.438,A 0.000,B 0.000,C 90.000,E1 294.823} C_DIS
LIN {X 0.145,Y -698.095,Z 796.435,A 0.000,B 0.000,C 90.000,E1 294.335} C_DIS
LIN {X -0.230,Y -698.058,Z 796.434,A 0.000,B 0.000,C 90.000,E1 294.131} C_DIS
LIN {X 0.008,Y -697.411,Z 796.431,A 0.000,B 0.000,C 90.000,E1 293.643} C_DIS
LIN {X 0.266,Y -696.715,Z 796.430,A 0.000,B 0.000,C 90.000,E1 293.387} C_DIS
LIN {X -0.265,Y -694.764,Z 796.428,A 0.000,B 0.000,C 90.000,E1 293.078} C_DIS
LIN {X -0.018,Y -693.210,Z 796.427,A 0.000,B 0.000,C 90.000,E1 292.823} C_DIS
LIN {X 0.104,Y -692.055,Z 796.426,A 0.000,B 0.000,C 90.000,E1 292.695} C_DIS
LIN {X -0.042,Y -690.282,Z 796.426,A 0.000,B 0.000,C 90.000,E1 292.589} C_DIS
LIN {X -0.045,Y -686.632,Z 796.424,A 0.000,B 0.000,C 90.000,E1 292.386} C_DIS
LIN {X 0.156,Y -683.285,Z 796.423,A 0.000,B 0.000,C 90.000,E1 292.206} C_DIS
LIN {X 0.055,Y -678.936,Z 796.423,A 0.000,B 0.000,C 90.000,E1 292.078} C_DIS
LIN {X 0.296,Y -673.521,Z 796.422,A 0.000,B 0.000,C 90.000,E1 291.897} C_DIS
LIN {X -0.138,Y -663.795,Z 796.421,A 0.000,B 0.000,C 90.000,E1 291.770} C_DIS
LIN {X 0.054,Y -653.285,Z 796.420,A 0.000,B 0.000,C 90.000,E1 291.589} C_DIS
LIN {X -0.004,Y -635.650,Z 796.418,A 0.000,B 0.000,C 90.000,E1 291.280} C_DIS
LIN {X -0.009,Y -615.157,Z 796.416,A 0.000,B 0.000,C 90.000,E1 290.844} C_DIS
LIN {X 0.132,Y -601.872,Z 796.414,A 0.000,B 0.000,C 90.000,E1 290.482} C_DIS
LIN {X -0.131,Y -585.093,Z 796.411,A 0.000,B 0.000,C 90.000,E1 289.993} C_DIS
LIN {X 0.036,Y -572.648,Z 796.408,A 0.000,B 0.000,C 90.000,E1 289.504} C_DIS
LIN {X -0.253,Y -567.502,Z 796.407,A 0.000,B 0.000,C 90.000,E1 289.268} C_DIS
LIN {X -0.224,Y -565.533,Z 796.406,A 0.000,B 0.000,C 90.000,E1 289.087} C_DIS
LIN {X 0.225,Y -563.795,Z 796.405,A 0.000,B 0.000,C 90.000,E1 288.906} C_DIS
LIN {X 0.092,Y -561.712,Z 796.403,A 0.000,B 0.000,C 90.000,E1 288.598} C_DIS
LIN {X -0.194,Y -560.978,Z 796.403,A 0.000,B 0.000,C 90.000,E1 288.489} C_DIS
LIN {X -0.003,Y -559.395,Z 796.400,A 0.000,B 0.000,C 90.000,E1 288.055} C_DIS
LIN {X 0.140,Y -557.820,Z 796.396,A 0.000,B 0.000,C 90.000,E1 287.347} C_DIS
LIN {X -0.116,Y -557.733,Z 796.395,A 0.000,B 0.000,C 90.000,E1 287.094} C_DIS
LIN {X -0.109,Y -557.969,Z 796.390,A 0.000,B 0.000,C 90.000,E1 286.260} C_DIS
LIN {X 0.302,Y -558.191,Z 796.390,A 0.000,B 0.000,C 90.000,E1 286.079} C_DIS
LIN {X 0.308,Y -559.873,Z 796.387,A 0.000,B 0.000,C 90.000,E1 285.662} C_DIS
LIN {X 0.047,Y -561.176,Z 796.384,A 0.000,B 0.000,C 90.000,E1 285.134} C_DIS
LIN {X -0.206,Y -562.089,Z 796.383,A 0.000,B 0.000,C 90.000,E1 284.883} C_DIS
LIN {X 0.094,Y -562.984,Z 796.380,A 0.000,B 0.000,C 90.000,E1 284.300} C_DIS
LIN {X 0.248,Y -563.040,Z 796.378,A 0.000,B 0.000,C 90.000,E1 284.008} C_DIS
LIN {X -0.086,Y -561.922,Z 796.372,A 0.000,B 0.000,C 90.000,E1 282.939} C_DIS
LIN {X 0.203,Y -561.195,Z 796.371,A 0.000,B 0.000,C 90.000,E1 282.771} C_DIS
LIN {X 0.068,Y -559.885,Z 796.370,A 0.000,B 0.000,C 90.000,E1 282.647} C_DIS
LIN {X -0.077,Y -557.824,Z 796.368,A 0.000,B 0.000,C 90.000,E1 282.299} C_DIS
LIN {X 0.206,Y -555.644,Z 796.365,A 0.000,B 0.000,C 90.000,E1 281.715} C_DIS
LIN {X 0.058,Y -554.668,Z 796.365,A 0.000,B 0.000,C 90.000,E1 281.591} C_DIS
LIN {X 0.215,Y -553.685,Z 796.363,A 0.000,B 0.000,C 90.000,E1 281.243} C_DIS
LIN {X -0.201,Y -553.327,Z 796.361,A 0.000,B 0.000,C 90.000,E1 281.007} C_DIS
LIN {X -0.078,Y -552.629,Z 796.360,A 0.000,B 0.000,C 90.000,E1 280.715} C_DIS
LIN {X 0.073,Y -551.841,Z 796.358,A 0.000,B 0.000,C 90.000,E1 280.489} C_DIS
LIN {X 0.119,Y -550.992,Z 796.347,A 0.000,B 0.000,C 90.000,E1 278.454} C_DIS
LIN {X -0.174,Y -550.900,Z 796.342,A 0.000,B 0.000,C 90.000,E1 277.644} C_DIS
LIN {X 0.181,Y -550.479,Z 796.336,A 0.000,B 0.000,C 90.000,E1 276.486} C_DIS
LIN {X -0.041,Y -549.837,Z 796.328,A 0.000,B 0.000,C 90.000,E1 275.106} C_DIS
LIN {X -0.270,Y -549.021,Z 796.321,A 0.000,B 0.000,C 90.000,E1 273.726} C_DIS
LIN {X 0.113,Y -547.710,Z 796.310,A 0.000,B 0.000,C 90.000,E1 271.718} C_DIS
LIN {X -0.159,Y -546.595,Z 796.300,A 0.000,B 0.000,C 90.000,E1 270.057} C_DIS
LIN {X 0.053,Y -545.604,Z 796.292,A 0.000,B 0.000,C 90.000,E1 268.625} C_DIS
LIN {X -0.192,Y -544.271,Z 796.281,A 0.000,B 0.000,C 90.000,E1 266.674} C_DIS
LIN {X 0.073,Y -543.069,Z 796.270,A 0.000,B 0.000,C 90.000,E1 264.666} C_DIS
LIN {X -0.221,Y -542.098,Z 796.263,A 0.000,B 0.000,C 90.000,E1 263.280} C_DIS
LIN {X -0.066,Y -541.424,Z 796.258,A 0.000,B 0.000,C 90.000,E1 262.413} C_DIS
LIN {X 0.216,Y -539.941,Z 796.248,A 0.000,B 0.000,C 90.000,E1 260.679} C_DIS
LIN {X -0.058,Y -538.648,Z 796.240,A 0.000,B 0.000,C 90.000,E1 259.285} C_DIS
LIN {X -0.193,Y -536.991,Z 796.231,A 0.000,B 0.000,C 90.000,E1 257.589} C_DIS
LIN {X -0.244,Y -535.281,Z 796.221,A 0.000,B 0.000,C 90.000,E1 255.880} C_DIS
LIN {X 0.274,Y -533.682,Z 796.214,A 0.000,B 0.000,C 90.000,E1 254.393} C_DIS
LIN {X -0.039,Y -531.344,Z 796.202,A 0.000,B 0.000,C 90.000,E1 252.417} C_DIS
LIN {X 0.058,Y -529.591,Z 796.194,A 0.000,B 0.000,C 90.000,E1 250.967} C_DIS
LIN {X 0.115,Y -527.695,Z 796.186,A 0.000,B 0.000,C 90.000,E1 249.518} C_DIS
LIN {X -0.178,Y -525.607,Z 796.178,A 0.000,B 0.000,C 90.000,E1 248.103} C_DIS
LIN {X 0.011,Y -523.889,Z 796.172,A 0.000,B 0.000,C 90.000,E1 246.922} C_DIS
LIN {X 0.002,Y -521.212,Z 796.162,A 0.000,B 0.000,C 90.000,E1 245.177} C_DIS
LIN {X -0.133,Y -519.329,Z 796.156,A 0.000,B 0.000,C 90.000,E1 244.024} C_DIS
LIN {X -0.291,Y -517.375,Z 796.149,A 0.000,B 0.000,C 90.000,E1 242.871} C_DIS
LIN {X -0.123,Y -514.835,Z 796.141,A 0.000,B 0.000,C 90.000,E1 241.385} C_DIS
LIN {X -0.115,Y -511.478,Z 796.131,A 0.000,B 0.000,C 90.000,E1 239.616} C_DIS
LIN {X -0.230,Y -509.763,Z 796.126,A 0.000,B 0.000,C 90.000,E1 238.742} C_DIS
LIN {X -0.035,Y -507.345,Z 796.120,A 0.000,B 0.000,C 90.000,E1 237.533} C_DIS
LIN {X 0.287,Y -504.260,Z 796.111,A 0.000,B 0.000,C 90.000,E1 236.008} C_DIS
LIN {X -0.149,Y -500.861,Z 796.103,A 0.000,B 0.000,C 90.000,E1 234.562} C_DIS
LIN {X 0.063,Y -497.918,Z 796.096,A 0.000,B 0.000,C 90.000,E1 233.336} C_DIS
LIN {X 0.096,Y -494.115,Z 796.088,A 0.000,B 0.000,C 90.000,E1 231.823} C_DIS
LIN {X 0.196,Y -488.200,Z 796.075,A 0.000,B 0.000,C 90.000,E1 229.380} C_DIS
LIN {X 0.111,Y -484.071,Z 796.064,A 0.000,B 0.000,C 90.000,E1 227.553} C_DIS
LIN {X -0.224,Y -480.797,Z 796.056,A 0.000,B 0.000,C 90.000,E1 226.053} C_DIS
LIN {X -0.165,Y -476.740,Z 796.045,A 0.000,B 0.000,C 90.000,E1 224.190} C_DIS
LIN {X -0.001,Y -471.285,Z 796.032,A 0.000,B 0.000,C 90.000,E1 221.676} C_DIS
LIN {X -0.102,Y -467.248,Z 796.021,A 0.000,B 0.000,C 90.000,E1 219.806} C_DIS
LIN {X -0.098,Y -464.661,Z 796.014,A 0.000,B 0.000,C 90.000,E1 218.543} C_DIS
LIN {X 0.116,Y -460.060,Z 796.002,A 0.000,B 0.000,C 90.000,E1 216.297} C_DIS
LIN {X 0.034,Y -455.365,Z 795.989,A 0.000,B 0.000,C 90.000,E1 214.072} C_DIS
LIN {X 0.114,Y -451.541,Z 795.979,A 0.000,B 0.000,C 90.000,E1 212.133} C_DIS
LIN {X 0.079,Y -447.005,Z 795.966,A 0.000,B 0.000,C 90.000,E1 209.873} C_DIS
LIN {X 0.249,Y -443.210,Z 795.955,A 0.000,B 0.000,C 90.000,E1 207.897} C_DIS
LIN {X 0.035,Y -440.790,Z 795.948,A 0.000,B 0.000,C 90.000,E1 206.616} C_DIS
LIN {X 0.041,Y -436.994,Z 795.937,A 0.000,B 0.000,C 90.000,E1 204.643} C_DIS
LIN {X 0.170,Y -433.170,Z 795.926,A 0.000,B 0.000,C 90.000,E1 202.642} C_DIS
LIN {X 0.038,Y -429.291,Z 795.915,A 0.000,B 0.000,C 90.000,E1 200.663} C_DIS
LIN {X -0.077,Y -425.485,Z 795.904,A 0.000,B 0.000,C 90.000,E1 198.671} C_DIS
LIN {X -0.114,Y -422.877,Z 795.896,A 0.000,B 0.000,C 90.000,E1 197.330} C_DIS
LIN {X -0.040,Y -420.276,Z 795.889,A 0.000,B 0.000,C 90.000,E1 195.969} C_DIS
LIN {X 0.002,Y -415.054,Z 795.874,A 0.000,B 0.000,C 90.000,E1 193.244} C_DIS
LIN {X -0.012,Y -411.852,Z 795.864,A 0.000,B 0.000,C 90.000,E1 191.535} C_DIS
LIN {X -0.186,Y -407.076,Z 795.849,A 0.000,B 0.000,C 90.000,E1 188.803} C_DIS
LIN {X -0.176,Y -403.967,Z 795.839,A 0.000,B 0.000,C 90.000,E1 187.068} C_DIS
LIN {X 0.112,Y -400.148,Z 795.828,A 0.000,B 0.000,C 90.000,E1 184.935} C_DIS
LIN {X -0.037,Y -394.445,Z 795.806,A 0.000,B 0.000,C 90.000,E1 181.088} C_DIS
LIN {X 0.015,Y -390.403,Z 795.786,A 0.000,B 0.000,C 90.000,E1 177.535} C_DIS
LIN {X -0.091,Y -388.150,Z 795.774,A 0.000,B 0.000,C 90.000,E1 175.412} C_DIS
LIN {X 0.126,Y -385.558,Z 795.761,A 0.000,B 0.000,C 90.000,E1 172.875} C_DIS
LIN {X 0.091,Y -383.845,Z 795.751,A 0.000,B 0.000,C 90.000,E1 171.084} C_DIS
LIN {X -0.197,Y -381.099,Z 795.733,A 0.000,B 0.000,C 90.000,E1 167.881} C_DIS
LIN {X 0.114,Y -378.901,Z 795.714,A 0.000,B 0.000,C 90.000,E1 164.574} C_DIS
LIN {X -0.035,Y -377.809,Z 795.702,A 0.000,B 0.000,C 90.000,E1 162.417} C_DIS
LIN {X -0.015,Y -376.860,Z 795.682,A 0.000,B 0.000,C 90.000,E1 158.773} C_DIS
LIN {X -0.042,Y -378.014,Z 795.650,A 0.000,B 0.000,C 90.000,E1 152.948} C_DIS
LIN {X 0.103,Y -380.130,Z 795.636,A 0.000,B 0.000,C 90.000,E1 150.383} C_DIS
LIN {X -0.130,Y -381.616,Z 795.630,A 0.000,B 0.000,C 90.000,E1 149.331} C_DIS
LIN {X -0.003,Y -384.228,Z 795.622,A 0.000,B 0.000,C 90.000,E1 147.867} C_DIS
LIN {X 0.006,Y -386.894,Z 795.616,A 0.000,B 0.000,C 90.000,E1 146.786} C_DIS
LIN {X -0.061,Y -390.019,Z 795.610,A 0.000,B 0.000,C 90.000,E1 145.722} C_DIS
LIN {X 0.192,Y -392.499,Z 795.606,A 0.000,B 0.000,C 90.000,E1 144.975} C_DIS
LIN {X -0.158,Y -395.040,Z 795.602,A 0.000,B 0.000,C 90.000,E1 144.402} C_DIS
LIN {X 0.016,Y -398.212,Z 795.599,A 0.000,B 0.000,C 90.000,E1 143.749} C_DIS
LIN {X 0.052,Y -402.099,Z 795.595,A 0.000,B 0.000,C 90.000,E1 143.084} C_DIS
LIN {X 0.088,Y -405.347,Z 795.592,A 0.000,B 0.000,C 90.000,E1 142.557} C_DIS
LIN {X -0.134,Y -411.463,Z 795.587,A 0.000,B 0.000,C 90.000,E1 141.743} C_DIS
LIN {X 0.084,Y -427.643,Z 795.576,A 0.000,B 0.000,C 90.000,E1 139.703} C_DIS
LIN {X 0.114,Y -441.808,Z 795.566,A 0.000,B 0.000,C 90.000,E1 137.919} C_DIS
LIN {X 0.168,Y -451.080,Z 795.560,A 0.000,B 0.000,C 90.000,E1 136.782} C_DIS
LIN {X 0.208,Y -458.750,Z 795.555,A 0.000,B 0.000,C 90.000,E1 135.810} C_DIS
LIN {X -0.013,Y -464.698,Z 795.550,A 0.000,B 0.000,C 90.000,E1 135.040} C_DIS
LIN {X -0.145,Y -471.602,Z 795.545,A 0.000,B 0.000,C 90.000,E1 134.109} C_DIS
LIN {X -0.139,Y -479.424,Z 795.539,A 0.000,B 0.000,C 90.000,E1 133.014} C_DIS
LIN {X 0.165,Y -484.652,Z 795.535,A 0.000,B 0.000,C 90.000,E1 132.204} C_DIS
LIN {X -0.056,Y -490.731,Z 795.530,A 0.000,B 0.000,C 90.000,E1 131.310} C_DIS
LIN {X 0.027,Y -495.548,Z 795.525,A 0.000,B 0.000,C 90.000,E1 130.539} C_DIS
LIN {X -0.099,Y -503.661,Z 795.518,A 0.000,B 0.000,C 90.000,E1 129.197} C_DIS
LIN {X -0.008,Y -507.112,Z 795.514,A 0.000,B 0.000,C 90.000,E1 128.588} C_DIS
LIN {X 0.219,Y -512.799,Z 795.509,A 0.000,B 0.000,C 90.000,E1 127.523} C_DIS
LIN {X -0.007,Y -517.328,Z 795.504,A 0.000,B 0.000,C 90.000,E1 126.664} C_DIS
LIN {X -0.186,Y -521.751,Z 795.499,A 0.000,B 0.000,C 90.000,E1 125.804} C_DIS
LIN {X -0.060,Y -526.669,Z 795.493,A 0.000,B 0.000,C 90.000,E1 124.771} C_DIS
LIN {X 0.115,Y -532.083,Z 795.486,A 0.000,B 0.000,C 90.000,E1 123.452} C_DIS
LIN {X -0.220,Y -535.561,Z 795.481,A 0.000,B 0.000,C 90.000,E1 122.625} C_DIS
LIN {X -0.066,Y -539.892,Z 795.475,A 0.000,B 0.000,C 90.000,E1 121.465} C_DIS
LIN {X -0.133,Y -543.990,Z 795.469,A 0.000,B 0.000,C 90.000,E1 120.335} C_DIS
LIN {X -0.143,Y -547.627,Z 795.462,A 0.000,B 0.000,C 90.000,E1 119.205} C_DIS
LIN {X 0.141,Y -551.867,Z 795.454,A 0.000,B 0.000,C 90.000,E1 117.769} C_DIS
LIN {X 0.172,Y -553.426,Z 795.451,A 0.000,B 0.000,C 90.000,E1 117.206} C_DIS
LIN {X 0.248,Y -555.423,Z 795.447,A 0.000,B 0.000,C 90.000,E1 116.360} C_DIS
LIN {X -0.117,Y -557.444,Z 795.440,A 0.000,B 0.000,C 90.000,E1 115.283} C_DIS
LIN {X -0.035,Y -558.379,Z 795.437,A 0.000,B 0.000,C 90.000,E1 114.719} C_DIS
LIN {X -0.153,Y -559.487,Z 795.433,A 0.000,B 0.000,C 90.000,E1 113.898} C_DIS
LIN {X 0.046,Y -560.678,Z 795.427,A 0.000,B 0.000,C 90.000,E1 112.770} C_DIS
LIN {X -0.159,Y -562.060,Z 795.419,A 0.000,B 0.000,C 90.000,E1 111.408} C_DIS
LIN {X 0.176,Y -563.230,Z 795.411,A 0.000,B 0.000,C 90.000,E1 109.993} C_DIS
LIN {X 0.017,Y -563.916,Z 795.405,A 0.000,B 0.000,C 90.000,E1 108.906} C_DIS
LIN {X -0.049,Y -564.984,Z 795.394,A 0.000,B 0.000,C 90.000,E1 106.985} C_DIS
LIN {X 0.067,Y -566.229,Z 795.382,A 0.000,B 0.000,C 90.000,E1 104.773} C_DIS
LIN {X -0.254,Y -567.483,Z 795.371,A 0.000,B 0.000,C 90.000,E1 102.883} C_DIS
LIN {X -0.100,Y -568.335,Z 795.365,A 0.000,B 0.000,C 90.000,E1 101.771} C_DIS
LIN {X 0.245,Y -569.408,Z 795.358,A 0.000,B 0.000,C 90.000,E1 100.366} C_DIS
LIN {X 0.040,Y -570.730,Z 795.349,A 0.000,B 0.000,C 90.000,E1 98.746} C_DIS
LIN {X -0.130,Y -571.838,Z 795.340,A 0.000,B 0.000,C 90.000,E1 97.125} C_DIS
LIN {X -0.088,Y -572.503,Z 795.333,A 0.000,B 0.000,C 90.000,E1 96.030} C_DIS
LIN {X 0.277,Y -573.473,Z 795.324,A 0.000,B 0.000,C 90.000,E1 94.359} C_DIS
LIN {X -0.107,Y -574.132,Z 795.317,A 0.000,B 0.000,C 90.000,E1 93.037} C_DIS
LIN {X -0.225,Y -574.958,Z 795.306,A 0.000,B 0.000,C 90.000,E1 91.146} C_DIS
LIN {X 0.095,Y -575.507,Z 795.297,A 0.000,B 0.000,C 90.000,E1 89.484} C_DIS
LIN {X 0.289,Y -575.984,Z 795.290,A 0.000,B 0.000,C 90.000,E1 88.108} C_DIS
LIN {X 0.071,Y -576.409,Z 795.281,A 0.000,B 0.000,C 90.000,E1 86.502} C_DIS
LIN {X 0.033,Y -576.881,Z 795.270,A 0.000,B 0.000,C 90.000,E1 84.609} C_DIS
LIN {X -0.097,Y -577.147,Z 795.261,A 0.000,B 0.000,C 90.000,E1 82.996} C_DIS
LIN {X -0.149,Y -577.444,Z 795.252,A 0.000,B 0.000,C 90.000,E1 81.376} C_DIS
LIN {X -0.099,Y -577.697,Z 795.243,A 0.000,B 0.000,C 90.000,E1 79.746} C_DIS
LIN {X -0.016,Y -577.855,Z 795.239,A 0.000,B 0.000,C 90.000,E1 78.926} C_DIS
LIN {X -0.179,Y -577.868,Z 795.231,A 0.000,B 0.000,C 90.000,E1 77.589} C_DIS
LIN {X 0.118,Y -577.797,Z 795.222,A 0.000,B 0.000,C 90.000,E1 75.936} C_DIS
LIN {X 0.062,Y -577.471,Z 795.211,A 0.000,B 0.000,C 90.000,E1 74.047} C_DIS
LIN {X -0.258,Y -577.256,Z 795.204,A 0.000,B 0.000,C 90.000,E1 72.725} C_DIS
LIN {X -0.203,Y -576.802,Z 795.195,A 0.000,B 0.000,C 90.000,E1 71.094} C_DIS
LIN {X 0.035,Y -576.170,Z 795.186,A 0.000,B 0.000,C 90.000,E1 69.444} C_DIS
LIN {X -0.116,Y -575.554,Z 795.178,A 0.000,B 0.000,C 90.000,E1 68.103} C_DIS
LIN {X -0.233,Y -574.667,Z 795.169,A 0.000,B 0.000,C 90.000,E1 66.485} C_DIS
LIN {X -0.134,Y -573.618,Z 795.160,A 0.000,B 0.000,C 90.000,E1 64.845} C_DIS
LIN {X 0.098,Y -572.563,Z 795.153,A 0.000,B 0.000,C 90.000,E1 63.461} C_DIS
LIN {X 0.214,Y -571.485,Z 795.147,A 0.000,B 0.000,C 90.000,E1 62.359} C_DIS
LIN {X -0.016,Y -570.555,Z 795.142,A 0.000,B 0.000,C 90.000,E1 61.563} C_DIS
LIN {X 0.076,Y -569.147,Z 795.136,A 0.000,B 0.000,C 90.000,E1 60.461} C_DIS
LIN {X -0.354,Y -567.517,Z 795.130,A 0.000,B 0.000,C 90.000,E1 59.410} C_DIS
LIN {X 0.157,Y -566.149,Z 795.125,A 0.000,B 0.000,C 90.000,E1 58.535} C_DIS
LIN {X -0.127,Y -564.630,Z 795.121,A 0.000,B 0.000,C 90.000,E1 57.740} C_DIS
LIN {X -0.125,Y -562.919,Z 795.116,A 0.000,B 0.000,C 90.000,E1 56.914} C_DIS
LIN {X -0.139,Y -561.039,Z 795.112,A 0.000,B 0.000,C 90.000,E1 56.087} C_DIS
LIN {X -0.085,Y -558.138,Z 795.105,A 0.000,B 0.000,C 90.000,E1 54.975} C_DIS
LIN {X 0.171,Y -555.786,Z 795.101,A 0.000,B 0.000,C 90.000,E1 54.116} C_DIS
LIN {X -0.001,Y -554.110,Z 795.098,A 0.000,B 0.000,C 90.000,E1 53.577} C_DIS
LIN {X -0.231,Y -551.216,Z 795.093,A 0.000,B 0.000,C 90.000,E1 52.763} C_DIS
LIN {X -0.105,Y -549.187,Z 795.090,A 0.000,B 0.000,C 90.000,E1 52.190} C_DIS
LIN {X 0.242,Y -545.182,Z 795.084,A 0.000,B 0.000,C 90.000,E1 51.170} C_DIS
LIN {X -0.105,Y -542.739,Z 795.081,A 0.000,B 0.000,C 90.000,E1 50.642} C_DIS
LIN {X 0.133,Y -539.303,Z 795.077,A 0.000,B 0.000,C 90.000,E1 49.908} C_DIS
LIN {X -0.253,Y -536.265,Z 795.074,A 0.000,B 0.000,C 90.000,E1 49.380} C_DIS
LIN {X 0.096,Y -533.063,Z 795.071,A 0.000,B 0.000,C 90.000,E1 48.771} C_DIS
LIN {X -0.166,Y -528.367,Z 795.067,A 0.000,B 0.000,C 90.000,E1 48.081} C_DIS
LIN {X 0.290,Y -524.428,Z 795.064,A 0.000,B 0.000,C 90.000,E1 47.472} C_DIS
LIN {X 0.057,Y -520.147,Z 795.061,A 0.000,B 0.000,C 90.000,E1 46.944} C_DIS
LIN {X 0.065,Y -515.319,Z 795.058,A 0.000,B 0.000,C 90.000,E1 46.377} C_DIS
LIN {X -0.006,Y -507.330,Z 795.053,A 0.000,B 0.000,C 90.000,E1 45.526} C_DIS
LIN {X 0.054,Y -500.096,Z 795.049,A 0.000,B 0.000,C 90.000,E1 44.838} C_DIS
LIN {X -0.030,Y -495.935,Z 795.047,A 0.000,B 0.000,C 90.000,E1 44.474} C_DIS
LIN {X -0.172,Y -491.449,Z 795.045,A 0.000,B 0.000,C 90.000,E1 44.109} C_DIS
LIN {X 0.119,Y -483.605,Z 795.042,A 0.000,B 0.000,C 90.000,E1 43.461} C_DIS
LIN {X -0.146,Y -478.840,Z 795.040,A 0.000,B 0.000,C 90.000,E1 43.137} C_DIS
LIN {X 0.061,Y -467.688,Z 795.035,A 0.000,B 0.000,C 90.000,E1 42.324} C_DIS
LIN {X 0.106,Y -448.377,Z 795.028,A 0.000,B 0.000,C 90.000,E1 40.987} C_DIS
LIN {X -0.022,Y -421.542,Z 795.017,A 0.000,B 0.000,C 90.000,E1 39.036} C_DIS
LIN {X -0.103,Y -407.619,Z 795.010,A 0.000,B 0.000,C 90.000,E1 37.890} C_DIS
LIN {X 0.178,Y -403.644,Z 795.008,A 0.000,B 0.000,C 90.000,E1 37.443} C_DIS
LIN {X 0.146,Y -403.606,Z 795.008,A 0.000,B 0.000,C 90.000,E1 37.443} C_DIS
LIN {X 0.037,Y -395.297,Z 794.983,A 0.000,B 0.000,C 90.000,E1 32.880} C_DIS
LIN {X -0.094,Y -395.230,Z 794.981,A 0.000,B 0.000,C 90.000,E1 32.546} C_DIS
LIN {X -0.127,Y -396.039,Z 794.967,A 0.000,B 0.000,C 90.000,E1 30.079} C_DIS
LIN {X -0.111,Y -397.475,Z 794.951,A 0.000,B 0.000,C 90.000,E1 27.257} C_DIS
LIN {X 0.056,Y -398.965,Z 794.938,A 0.000,B 0.000,C 90.000,E1 24.771} C_DIS
LIN {X -0.128,Y -401.276,Z 794.920,A 0.000,B 0.000,C 90.000,E1 21.642} C_DIS
LIN {X -0.056,Y -404.251,Z 794.903,A 0.000,B 0.000,C 90.000,E1 18.489} C_DIS
LIN {X 0.007,Y -408.681,Z 794.883,A 0.000,B 0.000,C 90.000,E1 15.009} C_DIS
LIN {X 0.104,Y -413.537,Z 794.866,A 0.000,B 0.000,C 90.000,E1 11.895} C_DIS
LIN {X 0.049,Y -417.136,Z 794.855,A 0.000,B 0.000,C 90.000,E1 9.849} C_DIS
LIN {X -0.002,Y -420.698,Z 794.843,A 0.000,B 0.000,C 90.000,E1 7.814} C_DIS
LIN {X -0.166,Y -423.736,Z 794.834,A 0.000,B 0.000,C 90.000,E1 6.144} C_DIS
LIN {X -0.131,Y -428.103,Z 794.821,A 0.000,B 0.000,C 90.000,E1 3.784} C_DIS
LIN {X -0.116,Y -431.921,Z 794.810,A 0.000,B 0.000,C 90.000,E1 1.776} C_DIS
LIN {X 0.165,Y -435.949,Z 794.799,A 0.000,B 0.000,C 90.000,E1 359.771} C_DIS
LIN {X 0.150,Y -441.713,Z 794.784,A 0.000,B 0.000,C 90.000,E1 357.135} C_DIS
LIN {X -0.222,Y -447.153,Z 794.772,A 0.000,B 0.000,C 90.000,E1 354.894} C_DIS
LIN {X 0.149,Y -451.081,Z 794.763,A 0.000,B 0.000,C 90.000,E1 353.223} C_DIS
LIN {X -0.095,Y -455.728,Z 794.752,A 0.000,B 0.000,C 90.000,E1 351.319} C_DIS
LIN {X -0.097,Y -460.438,Z 794.741,A 0.000,B 0.000,C 90.000,E1 349.398} C_DIS
LIN {X -0.072,Y -462.304,Z 794.738,A 0.000,B 0.000,C 90.000,E1 348.757} C_DIS
LIN {X -0.036,Y -464.672,Z 794.734,A 0.000,B 0.000,C 90.000,E1 348.117} C_DIS
LIN {X 0.100,Y -466.639,Z 794.732,A 0.000,B 0.000,C 90.000,E1 347.701} C_DIS
LIN {X -0.062,Y -470.124,Z 794.729,A 0.000,B 0.000,C 90.000,E1 347.229} C_DIS
LIN {X -0.017,Y -474.203,Z 794.726,A 0.000,B 0.000,C 90.000,E1 346.756} C_DIS
LIN {X 0.035,Y -480.715,Z 794.723,A 0.000,B 0.000,C 90.000,E1 346.172} C_DIS
LIN {X -0.251,Y -488.061,Z 794.720,A 0.000,B 0.000,C 90.000,E1 345.644} C_DIS
LIN {X -0.276,Y -506.814,Z 794.713,A 0.000,B 0.000,C 90.000,E1 344.338} C_DIS
LIN {X -0.188,Y -522.559,Z 794.707,A 0.000,B 0.000,C 90.000,E1 343.268} C_DIS
LIN {X -0.100,Y -535.092,Z 794.702,A 0.000,B 0.000,C 90.000,E1 342.417} C_DIS
LIN {X 0.112,Y -545.657,Z 794.698,A 0.000,B 0.000,C 90.000,E1 341.638} C_DIS
LIN {X -0.014,Y -552.997,Z 794.695,A 0.000,B 0.000,C 90.000,E1 341.094} C_DIS
LIN {X 0.118,Y -560.064,Z 794.692,A 0.000,B 0.000,C 90.000,E1 340.496} C_DIS
LIN {X 0.078,Y -565.376,Z 794.689,A 0.000,B 0.000,C 90.000,E1 340.007} C_DIS
LIN {X -0.275,Y -570.458,Z 794.686,A 0.000,B 0.000,C 90.000,E1 339.518} C_DIS
LIN {X -0.051,Y -575.232,Z 794.683,A 0.000,B 0.000,C 90.000,E1 338.954} C_DIS
LIN {X 0.259,Y -582.737,Z 794.678,A 0.000,B 0.000,C 90.000,E1 337.975} C_DIS
LIN {X 0.178,Y -588.600,Z 794.673,A 0.000,B 0.000,C 90.000,E1 337.177} C_DIS
LIN {X 0.340,Y -595.107,Z 794.668,A 0.000,B 0.000,C 90.000,E1 336.230} C_DIS
LIN {X -0.247,Y -601.984,Z 794.662,A 0.000,B 0.000,C 90.000,E1 335.229} C_DIS
LIN {X 0.079,Y -607.693,Z 794.657,A 0.000,B 0.000,C 90.000,E1 334.280} C_DIS
LIN {X -0.104,Y -614.615,Z 794.651,A 0.000,B 0.000,C 90.000,E1 333.127} C_DIS
LIN {X -0.163,Y -618.258,Z 794.647,A 0.000,B 0.000,C 90.000,E1 332.487} C_DIS
LIN {X 0.100,Y -623.923,Z 794.641,A 0.000,B 0.000,C 90.000,E1 331.435} C_DIS
LIN {X 0.137,Y -629.274,Z 794.636,A 0.000,B 0.000,C 90.000,E1 330.411} C_DIS
LIN {X -0.027,Y -633.195,Z 794.632,A 0.000,B 0.000,C 90.000,E1 329.665} C_DIS
LIN {X -0.108,Y -637.988,Z 794.626,A 0.000,B 0.000,C 90.000,E1 328.663} C_DIS
LIN {X -0.132,Y -642.451,Z 794.620,A 0.000,B 0.000,C 90.000,E1 327.661} C_DIS
LIN {X -0.165,Y -645.711,Z 794.616,A 0.000,B 0.000,C 90.000,E1 326.914} C_DIS
LIN {X -0.169,Y -648.705,Z 794.612,A 0.000,B 0.000,C 90.000,E1 326.167} C_DIS
LIN {X 0.199,Y -653.464,Z 794.605,A 0.000,B 0.000,C 90.000,E1 324.895} C_DIS
LIN {X -0.260,Y -657.761,Z 794.598,A 0.000,B 0.000,C 90.000,E1 323.703} C_DIS
LIN {X 0.230,Y -660.087,Z 794.594,A 0.000,B 0.000,C 90.000,E1 322.924} C_DIS
LIN {X -0.226,Y -663.166,Z 794.589,A 0.000,B 0.000,C 90.000,E1 321.984} C_DIS
LIN {X -0.228,Y -666.019,Z 794.583,A 0.000,B 0.000,C 90.000,E1 321.009} C_DIS
LIN {X -0.167,Y -667.408,Z 794.581,A 0.000,B 0.000,C 90.000,E1 320.517} C_DIS
LIN {X -0.111,Y -670.532,Z 794.574,A 0.000,B 0.000,C 90.000,E1 319.299} C_DIS
LIN {X 0.000,Y -673.485,Z 794.567,A 0.000,B 0.000,C 90.000,E1 318.081} C_DIS
LIN {X 0.040,Y -674.645,Z 794.565,A 0.000,B 0.000,C 90.000,E1 317.595} C_DIS
LIN {X 0.211,Y -677.132,Z 794.558,A 0.000,B 0.000,C 90.000,E1 316.377} C_DIS
LIN {X -0.085,Y -679.211,Z 794.551,A 0.000,B 0.000,C 90.000,E1 315.202} C_DIS
LIN {X -0.396,Y -680.846,Z 794.546,A 0.000,B 0.000,C 90.000,E1 314.271} C_DIS
LIN {X -0.159,Y -682.639,Z 794.539,A 0.000,B 0.000,C 90.000,E1 313.056} C_DIS
LIN {X 0.138,Y -684.257,Z 794.533,A 0.000,B 0.000,C 90.000,E1 311.838} C_DIS
LIN {X -0.102,Y -685.516,Z 794.527,A 0.000,B 0.000,C 90.000,E1 310.906} C_DIS
LIN {X -0.198,Y -686.849,Z 794.521,A 0.000,B 0.000,C 90.000,E1 309.725} C_DIS
LIN {X -0.216,Y -688.294,Z 794.513,A 0.000,B 0.000,C 90.000,E1 308.302} C_DIS
LIN {X -0.095,Y -689.640,Z 794.505,A 0.000,B 0.000,C 90.000,E1 306.870} C_DIS
LIN {X 0.012,Y -690.722,Z 794.498,A 0.000,B 0.000,C 90.000,E1 305.678} C_DIS
LIN {X 0.140,Y -691.608,Z 794.492,A 0.000,B 0.000,C 90.000,E1 304.485} C_DIS
LIN {X -0.211,Y -693.049,Z 794.481,A 0.000,B 0.000,C 90.000,E1 302.625} C_DIS
LIN {X 0.287,Y -694.642,Z 794.469,A 0.000,B 0.000,C 90.000,E1 300.463} C_DIS
LIN {X -0.285,Y -695.359,Z 794.463,A 0.000,B 0.000,C 90.000,E1 299.333} C_DIS
LIN {X 0.267,Y -696.286,Z 794.454,A 0.000,B 0.000,C 90.000,E1 297.641} C_DIS
LIN {X -0.148,Y -697.410,Z 794.443,A 0.000,B 0.000,C 90.000,E1 295.796} C_DIS
LIN {X 0.238,Y -698.115,Z 794.437,A 0.000,B 0.000,C 90.000,E1 294.591} C_DIS
LIN {X 0.127,Y -698.238,Z 794.434,A 0.000,B 0.000,C 90.000,E1 294.131} C_DIS
LIN {X -0.273,Y -697.518,Z 794.432,A 0.000,B 0.000,C 90.000,E1 293.695} C_DIS
LIN {X -0.293,Y -696.921,Z 794.430,A 0.000,B 0.000,C 90.000,E1 293.462} C_DIS
LIN {X -0.034,Y -695.603,Z 794.429,A 0.000,B 0.000,C 90.000,E1 293.206} C_DIS
LIN {X 0.340,Y -693.327,Z 794.427,A 0.000,B 0.000,C 90.000,E1 292.823} C_DIS
LIN {X 0.195,Y -692.270,Z 794.426,A 0.000,B 0.000,C 90.000,E1 292.717} C_DIS
LIN {X -0.323,Y -690.669,Z 794.426,A 0.000,B 0.000,C 90.000,E1 292.642} C_DIS
LIN {X 0.049,Y -686.821,Z 794.425,A 0.000,B 0.000,C 90.000,E1 292.408} C_DIS
LIN {X -0.108,Y -683.511,Z 794.424,A 0.000,B 0.000,C 90.000,E1 292.259} C_DIS
LIN {X 0.229,Y -681.385,Z 794.423,A 0.000,B 0.000,C 90.000,E1 292.153} C_DIS
LIN {X -0.031,Y -673.676,Z 794.422,A 0.000,B 0.000,C 90.000,E1 291.950} C_DIS
LIN {X 0.173,Y -663.900,Z 794.421,A 0.000,B 0.000,C 90.000,E1 291.770} C_DIS
LIN {X 0.255,Y -649.906,Z 794.420,A 0.000,B 0.000,C 90.000,E1 291.535} C_DIS
LIN {X 0.123,Y -632.717,Z 794.418,A 0.000,B 0.000,C 90.000,E1 291.227} C_DIS
LIN {X -0.060,Y -615.207,Z 794.416,A 0.000,B 0.000,C 90.000,E1 290.865} C_DIS
LIN {X 0.053,Y -605.631,Z 794.415,A 0.000,B 0.000,C 90.000,E1 290.610} C_DIS
LIN {X -0.186,Y -592.188,Z 794.412,A 0.000,B 0.000,C 90.000,E1 290.248} C_DIS
LIN {X 0.208,Y -581.982,Z 794.411,A 0.000,B 0.000,C 90.000,E1 289.885} C_DIS
LIN {X -0.182,Y -572.754,Z 794.409,A 0.000,B 0.000,C 90.000,E1 289.577} C_DIS
LIN {X -0.176,Y -569.796,Z 794.408,A 0.000,B 0.000,C 90.000,E1 289.450} C_DIS
LIN {X 0.138,Y -565.879,Z 794.407,A 0.000,B 0.000,C 90.000,E1 289.214} C_DIS
LIN {X 0.130,Y -562.513,Z 794.405,A 0.000,B 0.000,C 90.000,E1 288.960} C_DIS
LIN {X -0.185,Y -561.644,Z 794.405,A 0.000,B 0.000,C 90.000,E1 288.906} C_DIS
LIN {X -0.130,Y -559.972,Z 794.404,A 0.000,B 0.000,C 90.000,E1 288.671} C_DIS
LIN {X 0.032,Y -558.588,Z 794.402,A 0.000,B 0.000,C 90.000,E1 288.362} C_DIS
LIN {X 0.331,Y -557.457,Z 794.401,A 0.000,B 0.000,C 90.000,E1 288.055} C_DIS
LIN {X -0.218,Y -556.277,Z 794.398,A 0.000,B 0.000,C 90.000,E1 287.638} C_DIS
LIN {X 0.188,Y -555.270,Z 794.395,A 0.000,B 0.000,C 90.000,E1 287.040} C_DIS
LIN {X 0.011,Y -554.251,Z 794.389,A 0.000,B 0.000,C 90.000,E1 286.024} C_DIS
LIN {X 0.206,Y -554.234,Z 794.389,A 0.000,B 0.000,C 90.000,E1 285.969} C_DIS
LIN {X 0.164,Y -554.236,Z 794.389,A 0.000,B 0.000,C 90.000,E1 285.969} C_DIS
LIN {X 0.139,Y -554.395,Z 794.387,A 0.000,B 0.000,C 90.000,E1 285.662} C_DIS
LIN {X -0.277,Y -554.414,Z 794.386,A 0.000,B 0.000,C 90.000,E1 285.426} C_DIS
LIN {X -0.039,Y -554.659,Z 794.384,A 0.000,B 0.000,C 90.000,E1 285.134} C_DIS
LIN {X 0.227,Y -554.314,Z 794.383,A 0.000,B 0.000,C 90.000,E1 284.828} C_DIS
LIN {X -0.187,Y -554.242,Z 794.381,A 0.000,B 0.000,C 90.000,E1 284.592} C_DIS
LIN {X -0.306,Y -553.559,Z 794.376,A 0.000,B 0.000,C 90.000,E1 283.772} C_DIS
LIN {X -0.053,Y -553.277,Z 794.375,A 0.000,B 0.000,C 90.000,E1 283.467} C_DIS
LIN {X -0.229,Y -552.851,Z 794.370,A 0.000,B 0.000,C 90.000,E1 282.647} C_DIS
LIN {X 0.200,Y -551.532,Z 794.356,A 0.000,B 0.000,C 90.000,E1 280.084} C_DIS
LIN {X -0.034,Y -550.928,Z 794.342,A 0.000,B 0.000,C 90.000,E1 277.587} C_DIS
LIN {X -0.224,Y -550.490,Z 794.336,A 0.000,B 0.000,C 90.000,E1 276.486} C_DIS
LIN {X 0.057,Y -549.977,Z 794.330,A 0.000,B 0.000,C 90.000,E1 275.334} C_DIS
LIN {X -0.173,Y -549.177,Z 794.322,A 0.000,B 0.000,C 90.000,E1 273.955} C_DIS
LIN {X 0.257,Y -547.715,Z 794.309,A 0.000,B 0.000,C 90.000,E1 271.661} C_DIS
LIN {X -0.060,Y -546.768,Z 794.302,A 0.000,B 0.000,C 90.000,E1 270.286} C_DIS
LIN {X 0.196,Y -545.594,Z 794.292,A 0.000,B 0.000,C 90.000,E1 268.568} C_DIS
LIN {X -0.113,Y -544.439,Z 794.283,A 0.000,B 0.000,C 90.000,E1 266.906} C_DIS
LIN {X 0.193,Y -543.239,Z 794.272,A 0.000,B 0.000,C 90.000,E1 264.894} C_DIS
LIN {X -0.168,Y -542.508,Z 794.266,A 0.000,B 0.000,C 90.000,E1 263.799} C_DIS
LIN {X -0.003,Y -541.666,Z 794.259,A 0.000,B 0.000,C 90.000,E1 262.648} C_DIS
LIN {X -0.255,Y -540.178,Z 794.250,A 0.000,B 0.000,C 90.000,E1 260.971} C_DIS
LIN {X 0.103,Y -538.939,Z 794.242,A 0.000,B 0.000,C 90.000,E1 259.511} C_DIS
LIN {X 0.051,Y -537.011,Z 794.231,A 0.000,B 0.000,C 90.000,E1 257.521} C_DIS
LIN {X 0.011,Y -535.290,Z 794.221,A 0.000,B 0.000,C 90.000,E1 255.811} C_DIS
LIN {X -0.119,Y -533.698,Z 794.213,A 0.000,B 0.000,C 90.000,E1 254.393} C_DIS
LIN {X -0.174,Y -532.340,Z 794.207,A 0.000,B 0.000,C 90.000,E1 253.251} C_DIS
LIN {X -0.219,Y -530.648,Z 794.199,A 0.000,B 0.000,C 90.000,E1 251.819} C_DIS
LIN {X -0.146,Y -529.245,Z 794.193,A 0.000,B 0.000,C 90.000,E1 250.659} C_DIS
LIN {X -0.273,Y -527.694,Z 794.186,A 0.000,B 0.000,C 90.000,E1 249.518} C_DIS
LIN {X 0.119,Y -525.633,Z 794.178,A 0.000,B 0.000,C 90.000,E1 248.028} C_DIS
LIN {X 0.108,Y -523.879,Z 794.172,A 0.000,B 0.000,C 90.000,E1 246.869} C_DIS
LIN {X 0.158,Y -521.675,Z 794.164,A 0.000,B 0.000,C 90.000,E1 245.409} C_DIS
LIN {X -0.049,Y -519.301,Z 794.155,A 0.000,B 0.000,C 90.000,E1 243.973} C_DIS
LIN {X 0.025,Y -517.363,Z 794.149,A 0.000,B 0.000,C 90.000,E1 242.794} C_DIS
LIN {X 0.197,Y -514.810,Z 794.141,A 0.000,B 0.000,C 90.000,E1 241.307} C_DIS
LIN {X 0.208,Y -511.451,Z 794.131,A 0.000,B 0.000,C 90.000,E1 239.537} C_DIS
LIN {X 0.094,Y -509.731,Z 794.126,A 0.000,B 0.000,C 90.000,E1 238.663} C_DIS
LIN {X -0.037,Y -507.958,Z 794.121,A 0.000,B 0.000,C 90.000,E1 237.788} C_DIS
LIN {X -0.086,Y -504.240,Z 794.111,A 0.000,B 0.000,C 90.000,E1 236.008} C_DIS
LIN {X -0.114,Y -501.501,Z 794.104,A 0.000,B 0.000,C 90.000,E1 234.815} C_DIS
LIN {X -0.060,Y -499.346,Z 794.099,A 0.000,B 0.000,C 90.000,E1 233.909} C_DIS
LIN {X 0.002,Y -495.579,Z 794.091,A 0.000,B 0.000,C 90.000,E1 232.396} C_DIS
LIN {X -0.005,Y -490.302,Z 794.079,A 0.000,B 0.000,C 90.000,E1 230.275} C_DIS
LIN {X -0.213,Y -485.393,Z 794.068,A 0.000,B 0.000,C 90.000,E1 228.162} C_DIS
LIN {X 0.095,Y -480.738,Z 794.056,A 0.000,B 0.000,C 90.000,E1 225.972} C_DIS
LIN {X 0.150,Y -476.687,Z 794.045,A 0.000,B 0.000,C 90.000,E1 224.109} C_DIS
LIN {X -0.005,Y -471.228,Z 794.031,A 0.000,B 0.000,C 90.000,E1 221.634} C_DIS
LIN {X 0.202,Y -467.171,Z 794.021,A 0.000,B 0.000,C 90.000,E1 219.725} C_DIS
LIN {X 0.001,Y -463.264,Z 794.010,A 0.000,B 0.000,C 90.000,E1 217.855} C_DIS
LIN {X -0.236,Y -460.003,Z 794.002,A 0.000,B 0.000,C 90.000,E1 216.297} C_DIS
LIN {X -0.060,Y -455.302,Z 793.989,A 0.000,B 0.000,C 90.000,E1 214.040} C_DIS
LIN {X 0.149,Y -451.500,Z 793.978,A 0.000,B 0.000,C 90.000,E1 212.084} C_DIS
LIN {X -0.267,Y -446.971,Z 793.966,A 0.000,B 0.000,C 90.000,E1 209.873} C_DIS
LIN {X -0.151,Y -443.844,Z 793.957,A 0.000,B 0.000,C 90.000,E1 208.231} C_DIS
LIN {X 0.087,Y -440.763,Z 793.948,A 0.000,B 0.000,C 90.000,E1 206.565} C_DIS
LIN {X 0.098,Y -436.957,Z 793.937,A 0.000,B 0.000,C 90.000,E1 204.591} C_DIS
LIN {X -0.167,Y -433.179,Z 793.926,A 0.000,B 0.000,C 90.000,E1 202.642} C_DIS
LIN {X 0.106,Y -429.301,Z 793.915,A 0.000,B 0.000,C 90.000,E1 200.610} C_DIS
LIN {X 0.131,Y -425.480,Z 793.903,A 0.000,B 0.000,C 90.000,E1 198.598} C_DIS
LIN {X -0.039,Y -422.876,Z 793.896,A 0.000,B 0.000,C 90.000,E1 197.275} C_DIS
LIN {X 0.152,Y -420.269,Z 793.888,A 0.000,B 0.000,C 90.000,E1 195.898} C_DIS
LIN {X -0.181,Y -414.451,Z 793.871,A 0.000,B 0.000,C 90.000,E1 192.883} C_DIS
LIN {X 0.142,Y -410.603,Z 793.860,A 0.000,B 0.000,C 90.000,E1 190.782} C_DIS
LIN {X -0.100,Y -407.111,Z 793.849,A 0.000,B 0.000,C 90.000,E1 188.746} C_DIS
LIN {X -0.039,Y -404.009,Z 793.839,A 0.000,B 0.000,C 90.000,E1 187.004} C_DIS
LIN {X -0.198,Y -400.214,Z 793.827,A 0.000,B 0.000,C 90.000,E1 184.935} C_DIS
LIN {X 0.122,Y -395.002,Z 793.808,A 0.000,B 0.000,C 90.000,E1 181.375} C_DIS
LIN {X 0.193,Y -390.893,Z 793.788,A 0.000,B 0.000,C 90.000,E1 177.822} C_DIS
LIN {X 0.169,Y -389.033,Z 793.778,A 0.000,B 0.000,C 90.000,E1 176.045} C_DIS
LIN {X -0.160,Y -387.541,Z 793.770,A 0.000,B 0.000,C 90.000,E1 174.666} C_DIS
LIN {X 0.034,Y -385.049,Z 793.756,A 0.000,B 0.000,C 90.000,E1 172.129} C_DIS
LIN {X -0.119,Y -382.701,Z 793.742,A 0.000,B 0.000,C 90.000,E1 169.634} C_DIS
LIN {X -0.193,Y -380.756,Z 793.728,A 0.000,B 0.000,C 90.000,E1 167.117} C_DIS
LIN {X -0.151,Y -378.972,Z 793.712,A 0.000,B 0.000,C 90.000,E1 164.212} C_DIS
LIN {X 0.065,Y -377.957,Z 793.700,A 0.000,B 0.000,C 90.000,E1 162.000} C_DIS
LIN {X 0.080,Y -377.112,Z 793.680,A 0.000,B 0.000,C 90.000,E1 158.358} C_DIS
LIN {X 0.045,Y -378.478,Z 793.648,A 0.000,B 0.000,C 90.000,E1 152.538} C_DIS
LIN {X 0.027,Y -380.658,Z 793.633,A 0.000,B 0.000,C 90.000,E1 149.999} C_DIS
LIN {X -0.006,Y -382.217,Z 793.627,A 0.000,B 0.000,C 90.000,E1 148.918} C_DIS
LIN {X 0.133,Y -384.899,Z 793.619,A 0.000,B 0.000,C 90.000,E1 147.454} C_DIS
LIN {X -0.003,Y -386.645,Z 793.615,A 0.000,B 0.000,C 90.000,E1 146.755} C_DIS
LIN {X 0.200,Y -388.550,Z 793.611,A 0.000,B 0.000,C 90.000,E1 146.008} C_DIS
LIN {X -0.233,Y -391.275,Z 793.606,A 0.000,B 0.000,C 90.000,E1 145.182} C_DIS
LIN {X -0.079,Y -394.299,Z 793.602,A 0.000,B 0.000,C 90.000,E1 144.356} C_DIS
LIN {X 0.008,Y -397.297,Z 793.598,A 0.000,B 0.000,C 90.000,E1 143.703} C_DIS
LIN {X -0.098,Y -402.249,Z 793.594,A 0.000,B 0.000,C 90.000,E1 142.844} C_DIS
LIN {X -0.075,Y -405.613,Z 793.591,A 0.000,B 0.000,C 90.000,E1 142.316} C_DIS
LIN {X -0.010,Y -410.633,Z 793.587,A 0.000,B 0.000,C 90.000,E1 141.618} C_DIS
LIN {X -0.056,Y -426.734,Z 793.576,A 0.000,B 0.000,C 90.000,E1 139.622} C_DIS
LIN {X 0.117,Y -441.405,Z 793.566,A 0.000,B 0.000,C 90.000,E1 137.796} C_DIS
LIN {X -0.139,Y -450.824,Z 793.559,A 0.000,B 0.000,C 90.000,E1 136.701} C_DIS
LIN {X -0.084,Y -458.528,Z 793.554,A 0.000,B 0.000,C 90.000,E1 135.729} C_DIS
LIN {X -0.058,Y -463.166,Z 793.551,A 0.000,B 0.000,C 90.000,E1 135.121} C_DIS
LIN {X 0.063,Y -471.148,Z 793.545,A 0.000,B 0.000,C 90.000,E1 134.028} C_DIS
LIN {X 0.070,Y -479.076,Z 793.539,A 0.000,B 0.000,C 90.000,E1 132.933} C_DIS
LIN {X 0.298,Y -486.394,Z 793.533,A 0.000,B 0.000,C 90.000,E1 131.838} C_DIS
LIN {X -0.131,Y -492.348,Z 793.528,A 0.000,B 0.000,C 90.000,E1 130.987} C_DIS
LIN {X -0.122,Y -498.836,Z 793.522,A 0.000,B 0.000,C 90.000,E1 129.930} C_DIS
LIN {X -0.188,Y -504.273,Z 793.517,A 0.000,B 0.000,C 90.000,E1 129.036} C_DIS
LIN {X 0.198,Y -506.860,Z 793.514,A 0.000,B 0.000,C 90.000,E1 128.543} C_DIS
LIN {X 0.023,Y -512.615,Z 793.509,A 0.000,B 0.000,C 90.000,E1 127.523} C_DIS
LIN {X -0.332,Y -520.179,Z 793.500,A 0.000,B 0.000,C 90.000,E1 126.091} C_DIS
LIN {X 0.034,Y -526.603,Z 793.493,A 0.000,B 0.000,C 90.000,E1 124.739} C_DIS
LIN {X 0.217,Y -530.825,Z 793.487,A 0.000,B 0.000,C 90.000,E1 123.706} C_DIS
LIN {X 0.305,Y -535.485,Z 793.481,A 0.000,B 0.000,C 90.000,E1 122.546} C_DIS
LIN {X -0.283,Y -539.845,Z 793.475,A 0.000,B 0.000,C 90.000,E1 121.465} C_DIS
LIN {X 0.117,Y -543.968,Z 793.468,A 0.000,B 0.000,C 90.000,E1 120.285} C_DIS
LIN {X 0.114,Y -547.613,Z 793.462,A 0.000,B 0.000,C 90.000,E1 119.155} C_DIS
LIN {X 0.154,Y -551.060,Z 793.456,A 0.000,B 0.000,C 90.000,E1 118.025} C_DIS
LIN {X -0.052,Y -553.457,Z 793.451,A 0.000,B 0.000,C 90.000,E1 117.206} C_DIS
LIN {X 0.023,Y -555.467,Z 793.447,A 0.000,B 0.000,C 90.000,E1 116.360} C_DIS
LIN {X -0.342,Y -557.510,Z 793.440,A 0.000,B 0.000,C 90.000,E1 115.283} C_DIS
LIN {X 0.270,Y -558.829,Z 793.436,A 0.000,B 0.000,C 90.000,E1 114.387} C_DIS
LIN {X -0.151,Y -559.564,Z 793.433,A 0.000,B 0.000,C 90.000,E1 113.875} C_DIS
LIN {X -0.177,Y -560.729,Z 793.426,A 0.000,B 0.000,C 90.000,E1 112.770} C_DIS
LIN {X 0.140,Y -562.113,Z 793.419,A 0.000,B 0.000,C 90.000,E1 111.354} C_DIS
LIN {X 0.163,Y -563.087,Z 793.413,A 0.000,B 0.000,C 90.000,E1 110.248} C_DIS
LIN {X 0.192,Y -563.878,Z 793.406,A 0.000,B 0.000,C 90.000,E1 109.141} C_DIS
LIN {X 0.119,Y -565.010,Z 793.396,A 0.000,B 0.000,C 90.000,E1 107.221} C_DIS
LIN {X 0.235,Y -566.280,Z 793.384,A 0.000,B 0.000,C 90.000,E1 105.009} C_DIS
LIN {X -0.084,Y -567.566,Z 793.373,A 0.000,B 0.000,C 90.000,E1 103.119} C_DIS
LIN {X 0.252,Y -568.598,Z 793.365,A 0.000,B 0.000,C 90.000,E1 101.715} C_DIS
LIN {X 0.045,Y -569.705,Z 793.358,A 0.000,B 0.000,C 90.000,E1 100.366} C_DIS
LIN {X -0.154,Y -571.029,Z 793.349,A 0.000,B 0.000,C 90.000,E1 98.746} C_DIS
LIN {X 0.250,Y -572.141,Z 793.339,A 0.000,B 0.000,C 90.000,E1 97.068} C_DIS
LIN {X -0.212,Y -572.811,Z 793.333,A 0.000,B 0.000,C 90.000,E1 96.024} C_DIS
LIN {X 0.099,Y -573.783,Z 793.324,A 0.000,B 0.000,C 90.000,E1 94.359} C_DIS
LIN {X 0.294,Y -574.489,Z 793.317,A 0.000,B 0.000,C 90.000,E1 92.980} C_DIS
LIN {X 0.185,Y -575.295,Z 793.306,A 0.000,B 0.000,C 90.000,E1 91.088} C_DIS
LIN {X -0.061,Y -575.875,Z 793.297,A 0.000,B 0.000,C 90.000,E1 89.484} C_DIS
LIN {X 0.138,Y -576.348,Z 793.290,A 0.000,B 0.000,C 90.000,E1 88.108} C_DIS
LIN {X -0.072,Y -576.799,Z 793.281,A 0.000,B 0.000,C 90.000,E1 86.502} C_DIS
LIN {X -0.101,Y -577.236,Z 793.270,A 0.000,B 0.000,C 90.000,E1 84.609} C_DIS
LIN {X -0.153,Y -577.515,Z 793.261,A 0.000,B 0.000,C 90.000,E1 82.989} C_DIS
LIN {X -0.267,Y -577.818,Z 793.252,A 0.000,B 0.000,C 90.000,E1 81.376} C_DIS
LIN {X -0.211,Y -578.043,Z 793.243,A 0.000,B 0.000,C 90.000,E1 79.746} C_DIS
LIN {X 0.095,Y -578.185,Z 793.237,A 0.000,B 0.000,C 90.000,E1 78.634} C_DIS
LIN {X -0.282,Y -578.181,Z 793.231,A 0.000,B 0.000,C 90.000,E1 77.589} C_DIS
LIN {X 0.023,Y -578.084,Z 793.222,A 0.000,B 0.000,C 90.000,E1 75.936} C_DIS
LIN {X 0.132,Y -577.727,Z 793.211,A 0.000,B 0.000,C 90.000,E1 74.031} C_DIS
LIN {X 0.209,Y -577.487,Z 793.204,A 0.000,B 0.000,C 90.000,E1 72.670} C_DIS
LIN {X 0.073,Y -577.108,Z 793.196,A 0.000,B 0.000,C 90.000,E1 71.329} C_DIS
LIN {X 0.125,Y -576.462,Z 793.187,A 0.000,B 0.000,C 90.000,E1 69.699} C_DIS
LIN {X 0.185,Y -575.861,Z 793.180,A 0.000,B 0.000,C 90.000,E1 68.337} C_DIS
LIN {X -0.143,Y -574.970,Z 793.171,A 0.000,B 0.000,C 90.000,E1 66.741} C_DIS
LIN {X -0.248,Y -574.275,Z 793.165,A 0.000,B 0.000,C 90.000,E1 65.665} C_DIS
LIN {X 0.161,Y -573.505,Z 793.159,A 0.000,B 0.000,C 90.000,E1 64.537} C_DIS
LIN {X -0.128,Y -572.376,Z 793.151,A 0.000,B 0.000,C 90.000,E1 63.204} C_DIS
LIN {X -0.014,Y -571.227,Z 793.145,A 0.000,B 0.000,C 90.000,E1 62.103} C_DIS
LIN {X 0.082,Y -569.863,Z 793.139,A 0.000,B 0.000,C 90.000,E1 61.001} C_DIS
LIN {X -0.056,Y -568.308,Z 793.133,A 0.000,B 0.000,C 90.000,E1 59.921} C_DIS
LIN {X -0.010,Y -566.560,Z 793.127,A 0.000,B 0.000,C 90.000,E1 58.820} C_DIS
LIN {X 0.112,Y -564.494,Z 793.121,A 0.000,B 0.000,C 90.000,E1 57.709} C_DIS
LIN {X -0.190,Y -562.744,Z 793.116,A 0.000,B 0.000,C 90.000,E1 56.914} C_DIS
LIN {X -0.206,Y -560.815,Z 793.112,A 0.000,B 0.000,C 90.000,E1 56.087} C_DIS
LIN {X -0.155,Y -557.863,Z 793.105,A 0.000,B 0.000,C 90.000,E1 54.975} C_DIS
LIN {X 0.099,Y -555.449,Z 793.101,A 0.000,B 0.000,C 90.000,E1 54.116} C_DIS
LIN {X -0.074,Y -553.759,Z 793.098,A 0.000,B 0.000,C 90.000,E1 53.577} C_DIS
LIN {X 0.130,Y -550.784,Z 793.093,A 0.000,B 0.000,C 90.000,E1 52.718} C_DIS
LIN {X -0.185,Y -548.711,Z 793.090,A 0.000,B 0.000,C 90.000,E1 52.190} C_DIS
LIN {X 0.157,Y -544.620,Z 793.084,A 0.000,B 0.000,C 90.000,E1 51.170} C_DIS
LIN {X -0.193,Y -542.106,Z 793.081,A 0.000,B 0.000,C 90.000,E1 50.642} C_DIS
LIN {X 0.038,Y -538.577,Z 793.077,A 0.000,B 0.000,C 90.000,E1 49.908} C_DIS
LIN {X 0.055,Y -535.499,Z 793.074,A 0.000,B 0.000,C 90.000,E1 49.337} C_DIS
LIN {X 0.009,Y -532.230,Z 793.071,A 0.000,B 0.000,C 90.000,E1 48.771} C_DIS
LIN {X 0.324,Y -528.447,Z 793.068,A 0.000,B 0.000,C 90.000,E1 48.162} C_DIS
LIN {X -0.134,Y -524.328,Z 793.065,A 0.000,B 0.000,C 90.000,E1 47.634} C_DIS
LIN {X 0.010,Y -520.011,Z 793.062,A 0.000,B 0.000,C 90.000,E1 47.067} C_DIS
LIN {X 0.034,Y -515.182,Z 793.058,A 0.000,B 0.000,C 90.000,E1 46.500} C_DIS
LIN {X 0.131,Y -511.152,Z 793.056,A 0.000,B 0.000,C 90.000,E1 46.053} C_DIS
LIN {X 0.195,Y -505.709,Z 793.053,A 0.000,B 0.000,C 90.000,E1 45.486} C_DIS
LIN {X -0.242,Y -499.896,Z 793.050,A 0.000,B 0.000,C 90.000,E1 45.000} C_DIS
LIN {X 0.017,Y -495.727,Z 793.048,A 0.000,B 0.000,C 90.000,E1 44.595} C_DIS
LIN {X -0.203,Y -489.505,Z 793.045,A 0.000,B 0.000,C 90.000,E1 44.109} C_DIS
LIN {X 0.201,Y -481.700,Z 793.042,A 0.000,B 0.000,C 90.000,E1 43.461} C_DIS
LIN {X 0.103,Y -475.374,Z 793.039,A 0.000,B 0.000,C 90.000,E1 43.014} C_DIS
LIN {X -0.067,Y -465.789,Z 793.035,A 0.000,B 0.000,C 90.000,E1 42.366} C_DIS
LIN {X 0.079,Y -448.295,Z 793.029,A 0.000,B 0.000,C 90.000,E1 41.148} C_DIS
LIN {X 0.114,Y -419.640,Z 793.017,A 0.000,B 0.000,C 90.000,E1 39.036} C_DIS
LIN {X -0.184,Y -408.868,Z 793.012,A 0.000,B 0.000,C 90.000,E1 38.177} C_DIS
LIN {X 0.159,Y -404.059,Z 793.009,A 0.000,B 0.000,C 90.000,E1 37.649} C_DIS
LIN {X 0.128,Y -404.045,Z 793.009,A 0.000,B 0.000,C 90.000,E1 37.649} C_DIS
LIN {X -0.258,Y -395.665,Z 792.984,A 0.000,B 0.000,C 90.000,E1 33.166} C_DIS
LIN {X -0.047,Y -395.458,Z 792.983,A 0.000,B 0.000,C 90.000,E1 32.959} C_DIS
LIN {X 0.036,Y -396.235,Z 792.968,A 0.000,B 0.000,C 90.000,E1 30.285} C_DIS
LIN {X -0.160,Y -397.438,Z 792.955,A 0.000,B 0.000,C 90.000,E1 27.847} C_DIS
LIN {X 0.184,Y -398.862,Z 792.941,A 0.000,B 0.000,C 90.000,E1 25.335} C_DIS
LIN {X -0.079,Y -400.802,Z 792.925,A 0.000,B 0.000,C 90.000,E1 22.567} C_DIS
LIN {X 0.010,Y -403.195,Z 792.910,A 0.000,B 0.000,C 90.000,E1 19.758} C_DIS
LIN {X -0.133,Y -407.692,Z 792.889,A 0.000,B 0.000,C 90.000,E1 15.953} C_DIS
LIN {X 0.008,Y -412.320,Z 792.871,A 0.000,B 0.000,C 90.000,E1 12.827} C_DIS
LIN {X -0.080,Y -415.840,Z 792.860,A 0.000,B 0.000,C 90.000,E1 10.782} C_DIS
LIN {X -0.152,Y -418.782,Z 792.850,A 0.000,B 0.000,C 90.000,E1 9.086} C_DIS
LIN {X 0.111,Y -421.801,Z 792.841,A 0.000,B 0.000,C 90.000,E1 7.352} C_DIS
LIN {X -0.109,Y -424.222,Z 792.833,A 0.000,B 0.000,C 90.000,E1 6.030} C_DIS
LIN {X -0.114,Y -427.957,Z 792.822,A 0.000,B 0.000,C 90.000,E1 4.012} C_DIS
LIN {X -0.121,Y -431.763,Z 792.811,A 0.000,B 0.000,C 90.000,E1 2.007} C_DIS
LIN {X 0.165,Y -436.223,Z 792.799,A 0.000,B 0.000,C 90.000,E1 359.771} C_DIS
LIN {X 0.159,Y -441.958,Z 792.784,A 0.000,B 0.000,C 90.000,E1 357.135} C_DIS
LIN {X -0.206,Y -447.383,Z 792.772,A 0.000,B 0.000,C 90.000,E1 354.894} C_DIS
LIN {X -0.083,Y -452.076,Z 792.761,A 0.000,B 0.000,C 90.000,E1 352.932} C_DIS
LIN {X 0.148,Y -456.695,Z 792.750,A 0.000,B 0.000,C 90.000,E1 350.971} C_DIS
LIN {X 0.171,Y -461.416,Z 792.739,A 0.000,B 0.000,C 90.000,E1 349.050} C_DIS
LIN {X -0.251,Y -463.316,Z 792.736,A 0.000,B 0.000,C 90.000,E1 348.465} C_DIS
LIN {X 0.170,Y -465.115,Z 792.733,A 0.000,B 0.000,C 90.000,E1 347.937} C_DIS
LIN {X -0.202,Y -467.037,Z 792.731,A 0.000,B 0.000,C 90.000,E1 347.589} C_DIS
LIN {X 0.162,Y -469.048,Z 792.729,A 0.000,B 0.000,C 90.000,E1 347.229} C_DIS
LIN {X -0.212,Y -470.130,Z 792.728,A 0.000,B 0.000,C 90.000,E1 347.117} C_DIS
LIN {X -0.151,Y -474.618,Z 792.725,A 0.000,B 0.000,C 90.000,E1 346.589} C_DIS
LIN {X 0.200,Y -480.682,Z 792.722,A 0.000,B 0.000,C 90.000,E1 345.992} C_DIS
LIN {X -0.153,Y -489.848,Z 792.719,A 0.000,B 0.000,C 90.000,E1 345.338} C_DIS
LIN {X -0.145,Y -504.037,Z 792.713,A 0.000,B 0.000,C 90.000,E1 344.338} C_DIS
LIN {X -0.202,Y -524.586,Z 792.705,A 0.000,B 0.000,C 90.000,E1 342.960} C_DIS
LIN {X 0.260,Y -535.512,Z 792.701,A 0.000,B 0.000,C 90.000,E1 342.181} C_DIS
LIN {X -0.048,Y -546.121,Z 792.697,A 0.000,B 0.000,C 90.000,E1 341.456} C_DIS
LIN {X -0.089,Y -554.960,Z 792.693,A 0.000,B 0.000,C 90.000,E1 340.786} C_DIS
LIN {X -0.090,Y -560.509,Z 792.691,A 0.000,B 0.000,C 90.000,E1 340.315} C_DIS
LIN {X -0.210,Y -565.822,Z 792.688,A 0.000,B 0.000,C 90.000,E1 339.826} C_DIS
LIN {X 0.139,Y -570.866,Z 792.685,A 0.000,B 0.000,C 90.000,E1 339.263} C_DIS
LIN {X 0.139,Y -575.576,Z 792.682,A 0.000,B 0.000,C 90.000,E1 338.720} C_DIS
LIN {X -0.017,Y -582.045,Z 792.677,A 0.000,B 0.000,C 90.000,E1 337.922} C_DIS
LIN {X 0.118,Y -588.005,Z 792.673,A 0.000,B 0.000,C 90.000,E1 337.102} C_DIS
LIN {X -0.013,Y -595.423,Z 792.667,A 0.000,B 0.000,C 90.000,E1 336.049} C_DIS
LIN {X 0.197,Y -602.345,Z 792.661,A 0.000,B 0.000,C 90.000,E1 334.973} C_DIS
LIN {X -0.039,Y -608.841,Z 792.655,A 0.000,B 0.000,C 90.000,E1 333.948} C_DIS
LIN {X -0.188,Y -614.970,Z 792.650,A 0.000,B 0.000,C 90.000,E1 332.922} C_DIS
LIN {X -0.248,Y -619.331,Z 792.645,A 0.000,B 0.000,C 90.000,E1 332.153} C_DIS
LIN {X -0.269,Y -624.999,Z 792.640,A 0.000,B 0.000,C 90.000,E1 331.129} C_DIS
LIN {X 0.083,Y -630.360,Z 792.634,A 0.000,B 0.000,C 90.000,E1 330.078} C_DIS
LIN {X -0.097,Y -632.940,Z 792.631,A 0.000,B 0.000,C 90.000,E1 329.587} C_DIS
LIN {X 0.347,Y -637.195,Z 792.626,A 0.000,B 0.000,C 90.000,E1 328.663} C_DIS
LIN {X 0.269,Y -640.607,Z 792.622,A 0.000,B 0.000,C 90.000,E1 327.916} C_DIS
LIN {X 0.277,Y -645.036,Z 792.616,A 0.000,B 0.000,C 90.000,E1 326.914} C_DIS
LIN {X -0.269,Y -648.046,Z 792.612,A 0.000,B 0.000,C 90.000,E1 326.215} C_DIS
LIN {X 0.187,Y -651.973,Z 792.607,A 0.000,B 0.000,C 90.000,E1 325.182} C_DIS
LIN {X -0.294,Y -654.703,Z 792.603,A 0.000,B 0.000,C 90.000,E1 324.482} C_DIS
LIN {X -0.289,Y -658.154,Z 792.597,A 0.000,B 0.000,C 90.000,E1 323.497} C_DIS
LIN {X -0.289,Y -662.097,Z 792.590,A 0.000,B 0.000,C 90.000,E1 322.271} C_DIS
LIN {X 0.189,Y -665.734,Z 792.583,A 0.000,B 0.000,C 90.000,E1 321.009} C_DIS
LIN {X 0.237,Y -667.737,Z 792.579,A 0.000,B 0.000,C 90.000,E1 320.275} C_DIS
LIN {X 0.302,Y -670.352,Z 792.574,A 0.000,B 0.000,C 90.000,E1 319.299} C_DIS
LIN {X -0.022,Y -673.932,Z 792.566,A 0.000,B 0.000,C 90.000,E1 317.877} C_DIS
LIN {X 0.019,Y -675.030,Z 792.563,A 0.000,B 0.000,C 90.000,E1 317.391} C_DIS
LIN {X -0.335,Y -677.068,Z 792.558,A 0.000,B 0.000,C 90.000,E1 316.458} C_DIS
LIN {X -0.155,Y -679.194,Z 792.551,A 0.000,B 0.000,C 90.000,E1 315.243} C_DIS
LIN {X 0.017,Y -680.876,Z 792.546,A 0.000,B 0.000,C 90.000,E1 314.271} C_DIS
LIN {X -0.211,Y -682.702,Z 792.539,A 0.000,B 0.000,C 90.000,E1 313.095} C_DIS
LIN {X -0.411,Y -684.371,Z 792.533,A 0.000,B 0.000,C 90.000,E1 311.919} C_DIS
LIN {X -0.132,Y -685.639,Z 792.527,A 0.000,B 0.000,C 90.000,E1 310.943} C_DIS
LIN {X 0.224,Y -686.994,Z 792.521,A 0.000,B 0.000,C 90.000,E1 309.725} C_DIS
LIN {X 0.210,Y -688.446,Z 792.513,A 0.000,B 0.000,C 90.000,E1 308.302} C_DIS
LIN {X -0.264,Y -689.585,Z 792.506,A 0.000,B 0.000,C 90.000,E1 307.156} C_DIS
LIN {X 0.247,Y -690.669,Z 792.500,A 0.000,B 0.000,C 90.000,E1 305.931} C_DIS
LIN {X -0.029,Y -691.609,Z 792.493,A 0.000,B 0.000,C 90.000,E1 304.771} C_DIS
LIN {X 0.359,Y -692.813,Z 792.484,A 0.000,B 0.000,C 90.000,E1 303.086} C_DIS
LIN {X 0.110,Y -693.523,Z 792.479,A 0.000,B 0.000,C 90.000,E1 302.163} C_DIS
LIN {X -0.218,Y -694.829,Z 792.470,A 0.000,B 0.000,C 90.000,E1 300.541} C_DIS
LIN {X 0.166,Y -695.530,Z 792.463,A 0.000,B 0.000,C 90.000,E1 299.333} C_DIS
LIN {X -0.218,Y -696.433,Z 792.454,A 0.000,B 0.000,C 90.000,E1 297.719} C_DIS
LIN {X -0.317,Y -697.529,Z 792.443,A 0.000,B 0.000,C 90.000,E1 295.848} C_DIS
LIN {X -0.197,Y -698.150,Z 792.438,A 0.000,B 0.000,C 90.000,E1 294.899} C_DIS
LIN {X -0.333,Y -698.397,Z 792.434,A 0.000,B 0.000,C 90.000,E1 294.207} C_DIS
LIN {X 0.190,Y -697.677,Z 792.432,A 0.000,B 0.000,C 90.000,E1 293.695} C_DIS
LIN {X 0.171,Y -697.141,Z 792.430,A 0.000,B 0.000,C 90.000,E1 293.462} C_DIS
LIN {X 0.301,Y -696.577,Z 792.430,A 0.000,B 0.000,C 90.000,E1 293.334} C_DIS
LIN {X -0.106,Y -693.509,Z 792.427,A 0.000,B 0.000,C 90.000,E1 292.898} C_DIS
LIN {X 0.019,Y -692.546,Z 792.427,A 0.000,B 0.000,C 90.000,E1 292.770} C_DIS
LIN {X 0.138,Y -691.142,Z 792.426,A 0.000,B 0.000,C 90.000,E1 292.642} C_DIS
LIN {X -0.107,Y -687.239,Z 792.425,A 0.000,B 0.000,C 90.000,E1 292.461} C_DIS
LIN {X 0.133,Y -683.955,Z 792.424,A 0.000,B 0.000,C 90.000,E1 292.280} C_DIS
LIN {X 0.099,Y -682.127,Z 792.423,A 0.000,B 0.000,C 90.000,E1 292.206} C_DIS
LIN {X 0.023,Y -673.861,Z 792.422,A 0.000,B 0.000,C 90.000,E1 291.972} C_DIS
LIN {X -0.150,Y -660.448,Z 792.421,A 0.000,B 0.000,C 90.000,E1 291.770} C_DIS
LIN {X -0.038,Y -643.101,Z 792.419,A 0.000,B 0.000,C 90.000,E1 291.461} C_DIS
LIN {X -0.234,Y -632.930,Z 792.418,A 0.000,B 0.000,C 90.000,E1 291.280} C_DIS
LIN {X 0.114,Y -615.248,Z 792.416,A 0.000,B 0.000,C 90.000,E1 290.865} C_DIS
LIN {X 0.194,Y -605.500,Z 792.415,A 0.000,B 0.000,C 90.000,E1 290.610} C_DIS
LIN {X -0.087,Y -591.695,Z 792.412,A 0.000,B 0.000,C 90.000,E1 290.248} C_DIS
LIN {X -0.173,Y -581.503,Z 792.411,A 0.000,B 0.000,C 90.000,E1 289.939} C_DIS
LIN {X 0.001,Y -572.063,Z 792.409,A 0.000,B 0.000,C 90.000,E1 289.577} C_DIS
LIN {X -0.159,Y -567.487,Z 792.408,A 0.000,B 0.000,C 90.000,E1 289.396} C_DIS
LIN {X -0.215,Y -564.049,Z 792.407,A 0.000,B 0.000,C 90.000,E1 289.214} C_DIS
LIN {X 0.048,Y -561.036,Z 792.405,A 0.000,B 0.000,C 90.000,E1 288.960} C_DIS
LIN {X 0.088,Y -558.437,Z 792.403,A 0.000,B 0.000,C 90.000,E1 288.598} C_DIS
LIN {X -0.092,Y -556.641,Z 792.401,A 0.000,B 0.000,C 90.000,E1 288.181} C_DIS
LIN {X -0.093,Y -555.649,Z 792.399,A 0.000,B 0.000,C 90.000,E1 287.764} C_DIS
LIN {X -0.221,Y -554.732,Z 792.396,A 0.000,B 0.000,C 90.000,E1 287.221} C_DIS
LIN {X -0.086,Y -553.885,Z 792.391,A 0.000,B 0.000,C 90.000,E1 286.370} C_DIS
LIN {X 0.070,Y -553.099,Z 792.379,A 0.000,B 0.000,C 90.000,E1 284.120} C_DIS
LIN {X -0.048,Y -552.249,Z 792.368,A 0.000,B 0.000,C 90.000,E1 282.175} C_DIS
LIN {X 0.245,Y -551.443,Z 792.355,A 0.000,B 0.000,C 90.000,E1 279.905} C_DIS
LIN {X -0.110,Y -550.968,Z 792.343,A 0.000,B 0.000,C 90.000,E1 277.701} C_DIS
LIN {X 0.141,Y -550.724,Z 792.338,A 0.000,B 0.000,C 90.000,E1 276.834} C_DIS
LIN {X -0.073,Y -550.042,Z 792.330,A 0.000,B 0.000,C 90.000,E1 275.454} C_DIS
LIN {X -0.253,Y -549.249,Z 792.323,A 0.000,B 0.000,C 90.000,E1 274.069} C_DIS
LIN {X 0.178,Y -547.798,Z 792.310,A 0.000,B 0.000,C 90.000,E1 271.776} C_DIS
LIN {X -0.139,Y -546.851,Z 792.302,A 0.000,B 0.000,C 90.000,E1 270.401} C_DIS
LIN {X 0.120,Y -545.692,Z 792.293,A 0.000,B 0.000,C 90.000,E1 268.682} C_DIS
LIN {X -0.186,Y -544.531,Z 792.283,A 0.000,B 0.000,C 90.000,E1 267.020} C_DIS
LIN {X 0.125,Y -543.336,Z 792.272,A 0.000,B 0.000,C 90.000,E1 265.008} C_DIS
LIN {X -0.219,Y -542.406,Z 792.265,A 0.000,B 0.000,C 90.000,E1 263.628} C_DIS
LIN {X 0.011,Y -541.515,Z 792.258,A 0.000,B 0.000,C 90.000,E1 262.470} C_DIS
LIN {X 0.225,Y -540.284,Z 792.250,A 0.000,B 0.000,C 90.000,E1 261.027} C_DIS
LIN {X -0.041,Y -539.075,Z 792.242,A 0.000,B 0.000,C 90.000,E1 259.634} C_DIS
LIN {X -0.100,Y -537.156,Z 792.231,A 0.000,B 0.000,C 90.000,E1 257.645} C_DIS
LIN {X -0.145,Y -535.474,Z 792.222,A 0.000,B 0.000,C 90.000,E1 255.936} C_DIS
LIN {X -0.089,Y -533.549,Z 792.212,A 0.000,B 0.000,C 90.000,E1 254.212} C_DIS
LIN {X 0.104,Y -531.205,Z 792.201,A 0.000,B 0.000,C 90.000,E1 252.181} C_DIS
LIN {X 0.194,Y -529.474,Z 792.193,A 0.000,B 0.000,C 90.000,E1 250.732} C_DIS
LIN {X 0.247,Y -527.898,Z 792.187,A 0.000,B 0.000,C 90.000,E1 249.571} C_DIS
LIN {X -0.038,Y -525.846,Z 792.179,A 0.000,B 0.000,C 90.000,E1 248.156} C_DIS
LIN {X 0.158,Y -524.117,Z 792.172,A 0.000,B 0.000,C 90.000,E1 246.975} C_DIS
LIN {X 0.007,Y -521.917,Z 792.164,A 0.000,B 0.000,C 90.000,E1 245.537} C_DIS
LIN {X 0.031,Y -519.549,Z 792.156,A 0.000,B 0.000,C 90.000,E1 244.076} C_DIS
LIN {X 0.009,Y -517.111,Z 792.148,A 0.000,B 0.000,C 90.000,E1 242.615} C_DIS
LIN {X 0.059,Y -515.051,Z 792.141,A 0.000,B 0.000,C 90.000,E1 241.435} C_DIS
LIN {X 0.079,Y -511.718,Z 792.132,A 0.000,B 0.000,C 90.000,E1 239.665} C_DIS
LIN {X 0.041,Y -509.435,Z 792.125,A 0.000,B 0.000,C 90.000,E1 238.486} C_DIS
LIN {X -0.157,Y -508.273,Z 792.122,A 0.000,B 0.000,C 90.000,E1 237.916} C_DIS
LIN {X 0.225,Y -504.542,Z 792.112,A 0.000,B 0.000,C 90.000,E1 236.087} C_DIS
LIN {X 0.196,Y -501.827,Z 792.105,A 0.000,B 0.000,C 90.000,E1 234.895} C_DIS
LIN {X 0.252,Y -499.683,Z 792.100,A 0.000,B 0.000,C 90.000,E1 233.989} C_DIS
LIN {X 0.315,Y -495.932,Z 792.092,A 0.000,B 0.000,C 90.000,E1 232.477} C_DIS
LIN {X 0.311,Y -490.634,Z 792.080,A 0.000,B 0.000,C 90.000,E1 230.356} C_DIS
LIN {X -0.075,Y -485.008,Z 792.066,A 0.000,B 0.000,C 90.000,E1 227.957} C_DIS
LIN {X -0.263,Y -481.012,Z 792.056,A 0.000,B 0.000,C 90.000,E1 226.134} C_DIS
LIN {X 0.020,Y -477.630,Z 792.048,A 0.000,B 0.000,C 90.000,E1 224.555} C_DIS
LIN {X -0.085,Y -476.264,Z 792.044,A 0.000,B 0.000,C 90.000,E1 223.947} C_DIS
LIN {X -0.025,Y -471.522,Z 792.032,A 0.000,B 0.000,C 90.000,E1 221.757} C_DIS
LIN {X 0.040,Y -468.794,Z 792.025,A 0.000,B 0.000,C 90.000,E1 220.496} C_DIS
LIN {X -0.055,Y -466.799,Z 792.020,A 0.000,B 0.000,C 90.000,E1 219.564} C_DIS
LIN {X 0.059,Y -463.560,Z 792.011,A 0.000,B 0.000,C 90.000,E1 217.971} C_DIS
LIN {X 0.114,Y -460.300,Z 792.002,A 0.000,B 0.000,C 90.000,E1 216.377} C_DIS
LIN {X 0.024,Y -454.945,Z 791.988,A 0.000,B 0.000,C 90.000,E1 213.833} C_DIS
LIN {X 0.132,Y -451.776,Z 791.979,A 0.000,B 0.000,C 90.000,E1 212.212} C_DIS
LIN {X 0.031,Y -447.914,Z 791.968,A 0.000,B 0.000,C 90.000,E1 210.285} C_DIS
LIN {X -0.156,Y -444.144,Z 791.957,A 0.000,B 0.000,C 90.000,E1 208.359} C_DIS
LIN {X 0.086,Y -441.067,Z 791.948,A 0.000,B 0.000,C 90.000,E1 206.693} C_DIS
LIN {X 0.106,Y -437.264,Z 791.937,A 0.000,B 0.000,C 90.000,E1 204.719} C_DIS
LIN {X -0.150,Y -433.494,Z 791.926,A 0.000,B 0.000,C 90.000,E1 202.770} C_DIS
LIN {X -0.055,Y -429.002,Z 791.914,A 0.000,B 0.000,C 90.000,E1 200.429} C_DIS
LIN {X -0.036,Y -425.147,Z 791.902,A 0.000,B 0.000,C 90.000,E1 198.417} C_DIS
LIN {X 0.007,Y -423.226,Z 791.897,A 0.000,B 0.000,C 90.000,E1 197.402} C_DIS
LIN {X -0.024,Y -419.951,Z 791.887,A 0.000,B 0.000,C 90.000,E1 195.717} C_DIS
LIN {X -0.104,Y -414.796,Z 791.872,A 0.000,B 0.000,C 90.000,E1 193.008} C_DIS
LIN {X -0.126,Y -411.572,Z 791.863,A 0.000,B 0.000,C 90.000,E1 191.299} C_DIS
LIN {X 0.072,Y -407.408,Z 791.849,A 0.000,B 0.000,C 90.000,E1 188.859} C_DIS
LIN {X 0.083,Y -404.389,Z 791.840,A 0.000,B 0.000,C 90.000,E1 187.125} C_DIS
LIN {X -0.037,Y -400.021,Z 791.826,A 0.000,B 0.000,C 90.000,E1 184.702} C_DIS
LIN {X -0.150,Y -394.861,Z 791.807,A 0.000,B 0.000,C 90.000,E1 181.203} C_DIS
LIN {X 0.000,Y -391.146,Z 791.789,A 0.000,B 0.000,C 90.000,E1 177.993} C_DIS
LIN {X -0.015,Y -389.349,Z 791.779,A 0.000,B 0.000,C 90.000,E1 176.216} C_DIS
LIN {X 0.049,Y -387.891,Z 791.771,A 0.000,B 0.000,C 90.000,E1 174.780} C_DIS
LIN {X -0.126,Y -385.372,Z 791.757,A 0.000,B 0.000,C 90.000,E1 172.299} C_DIS
LIN {X -0.033,Y -383.998,Z 791.749,A 0.000,B 0.000,C 90.000,E1 170.849} C_DIS
LIN {X 0.152,Y -381.662,Z 791.733,A 0.000,B 0.000,C 90.000,E1 167.937} C_DIS
LIN {X 0.132,Y -379.967,Z 791.719,A 0.000,B 0.000,C 90.000,E1 165.408} C_DIS
LIN {X -0.111,Y -378.652,Z 791.705,A 0.000,B 0.000,C 90.000,E1 162.906} C_DIS
LIN {X -0.162,Y -377.722,Z 791.691,A 0.000,B 0.000,C 90.000,E1 160.369} C_DIS
LIN {X 0.018,Y -377.371,Z 791.677,A 0.000,B 0.000,C 90.000,E1 157.794} C_DIS
LIN {X -0.134,Y -378.838,Z 791.646,A 0.000,B 0.000,C 90.000,E1 152.359} C_DIS
LIN {X 0.225,Y -380.595,Z 791.634,A 0.000,B 0.000,C 90.000,E1 150.127} C_DIS
LIN {X -0.187,Y -382.607,Z 791.626,A 0.000,B 0.000,C 90.000,E1 148.742} C_DIS
LIN {X -0.199,Y -384.420,Z 791.620,A 0.000,B 0.000,C 90.000,E1 147.661} C_DIS
LIN {X 0.228,Y -388.628,Z 791.610,A 0.000,B 0.000,C 90.000,E1 145.801} C_DIS
LIN {X 0.124,Y -390.727,Z 791.606,A 0.000,B 0.000,C 90.000,E1 145.102} C_DIS
LIN {X 0.039,Y -393.233,Z 791.602,A 0.000,B 0.000,C 90.000,E1 144.402} C_DIS
LIN {X -0.026,Y -396.313,Z 791.598,A 0.000,B 0.000,C 90.000,E1 143.703} C_DIS
LIN {X -0.097,Y -400.987,Z 791.594,A 0.000,B 0.000,C 90.000,E1 142.844} C_DIS
LIN {X -0.006,Y -404.118,Z 791.591,A 0.000,B 0.000,C 90.000,E1 142.316} C_DIS
LIN {X 0.070,Y -408.637,Z 791.587,A 0.000,B 0.000,C 90.000,E1 141.662} C_DIS
LIN {X 0.232,Y -426.187,Z 791.575,A 0.000,B 0.000,C 90.000,E1 139.461} C_DIS
LIN {X 0.124,Y -442.047,Z 791.564,A 0.000,B 0.000,C 90.000,E1 137.553} C_DIS
LIN {X -0.081,Y -451.533,Z 791.558,A 0.000,B 0.000,C 90.000,E1 136.458} C_DIS
LIN {X -0.002,Y -457.962,Z 791.554,A 0.000,B 0.000,C 90.000,E1 135.648} C_DIS
LIN {X 0.001,Y -461.526,Z 791.551,A 0.000,B 0.000,C 90.000,E1 135.202} C_DIS
LIN {X 0.142,Y -470.825,Z 791.544,A 0.000,B 0.000,C 90.000,E1 133.947} C_DIS
LIN {X 0.145,Y -478.834,Z 791.538,A 0.000,B 0.000,C 90.000,E1 132.852} C_DIS
LIN {X 0.295,Y -486.358,Z 791.532,A 0.000,B 0.000,C 90.000,E1 131.757} C_DIS
LIN {X 0.018,Y -491.460,Z 791.528,A 0.000,B 0.000,C 90.000,E1 131.024} C_DIS
LIN {X 0.151,Y -499.962,Z 791.520,A 0.000,B 0.000,C 90.000,E1 129.644} C_DIS
LIN {X 0.102,Y -505.414,Z 791.515,A 0.000,B 0.000,C 90.000,E1 128.749} C_DIS
LIN {X -0.094,Y -511.252,Z 791.510,A 0.000,B 0.000,C 90.000,E1 127.729} C_DIS
LIN {X -0.068,Y -513.638,Z 791.507,A 0.000,B 0.000,C 90.000,E1 127.282} C_DIS
LIN {X 0.189,Y -520.427,Z 791.500,A 0.000,B 0.000,C 90.000,E1 125.931} C_DIS
LIN {X -0.304,Y -526.219,Z 791.493,A 0.000,B 0.000,C 90.000,E1 124.818} C_DIS
LIN {X -0.125,Y -530.499,Z 791.488,A 0.000,B 0.000,C 90.000,E1 123.785} C_DIS
LIN {X -0.038,Y -535.177,Z 791.481,A 0.000,B 0.000,C 90.000,E1 122.625} C_DIS
LIN {X 0.111,Y -538.529,Z 791.477,A 0.000,B 0.000,C 90.000,E1 121.750} C_DIS
LIN {X 0.309,Y -542.689,Z 791.470,A 0.000,B 0.000,C 90.000,E1 120.590} C_DIS
LIN {X -0.207,Y -545.603,Z 791.465,A 0.000,B 0.000,C 90.000,E1 119.795} C_DIS
LIN {X 0.282,Y -549.160,Z 791.459,A 0.000,B 0.000,C 90.000,E1 118.615} C_DIS
LIN {X 0.312,Y -551.702,Z 791.455,A 0.000,B 0.000,C 90.000,E1 117.769} C_DIS
LIN {X -0.151,Y -553.315,Z 791.451,A 0.000,B 0.000,C 90.000,E1 117.257} C_DIS
LIN {X -0.081,Y -555.364,Z 791.447,A 0.000,B 0.000,C 90.000,E1 116.411} C_DIS
LIN {X -0.238,Y -556.997,Z 791.442,A 0.000,B 0.000,C 90.000,E1 115.591} C_DIS
LIN {X 0.135,Y -558.409,Z 791.437,A 0.000,B 0.000,C 90.000,E1 114.719} C_DIS
LIN {X 0.017,Y -559.548,Z 791.433,A 0.000,B 0.000,C 90.000,E1 113.898} C_DIS
LIN {X 0.217,Y -560.716,Z 791.427,A 0.000,B 0.000,C 90.000,E1 112.770} C_DIS
LIN {X 0.012,Y -562.129,Z 791.419,A 0.000,B 0.000,C 90.000,E1 111.408} C_DIS
LIN {X 0.350,Y -563.347,Z 791.411,A 0.000,B 0.000,C 90.000,E1 109.993} C_DIS
LIN {X 0.193,Y -564.100,Z 791.405,A 0.000,B 0.000,C 90.000,E1 108.906} C_DIS
LIN {X -0.020,Y -565.132,Z 791.396,A 0.000,B 0.000,C 90.000,E1 107.275} C_DIS
LIN {X 0.161,Y -566.094,Z 791.387,A 0.000,B 0.000,C 90.000,E1 105.607} C_DIS
LIN {X 0.050,Y -567.005,Z 791.379,A 0.000,B 0.000,C 90.000,E1 104.245} C_DIS
LIN {X 0.127,Y -568.213,Z 791.370,A 0.000,B 0.000,C 90.000,E1 102.591} C_DIS
LIN {X -0.094,Y -569.956,Z 791.358,A 0.000,B 0.000,C 90.000,E1 100.423} C_DIS
LIN {X -0.292,Y -571.280,Z 791.349,A 0.000,B 0.000,C 90.000,E1 98.803} C_DIS
LIN {X 0.115,Y -572.408,Z 791.340,A 0.000,B 0.000,C 90.000,E1 97.125} C_DIS
LIN {X 0.166,Y -573.092,Z 791.334,A 0.000,B 0.000,C 90.000,E1 96.030} C_DIS
LIN {X -0.164,Y -573.872,Z 791.326,A 0.000,B 0.000,C 90.000,E1 94.702} C_DIS
LIN {X -0.145,Y -574.493,Z 791.320,A 0.000,B 0.000,C 90.000,E1 93.612} C_DIS
LIN {X -0.114,Y -575.029,Z 791.314,A 0.000,B 0.000,C 90.000,E1 92.522} C_DIS
LIN {X 0.070,Y -575.618,Z 791.306,A 0.000,B 0.000,C 90.000,E1 91.146} C_DIS
LIN {X -0.018,Y -576.334,Z 791.296,A 0.000,B 0.000,C 90.000,E1 89.255} C_DIS
LIN {X 0.190,Y -576.792,Z 791.288,A 0.000,B 0.000,C 90.000,E1 87.879} C_DIS
LIN {X -0.167,Y -577.171,Z 791.281,A 0.000,B 0.000,C 90.000,E1 86.560} C_DIS
LIN {X -0.186,Y -577.581,Z 791.270,A 0.000,B 0.000,C 90.000,E1 84.666} C_DIS
LIN {X -0.299,Y -577.872,Z 791.261,A 0.000,B 0.000,C 90.000,E1 83.053} C_DIS
LIN {X 0.238,Y -578.165,Z 791.252,A 0.000,B 0.000,C 90.000,E1 81.376} C_DIS
LIN {X -0.266,Y -578.385,Z 791.243,A 0.000,B 0.000,C 90.000,E1 79.803} C_DIS
LIN {X 0.152,Y -578.509,Z 791.236,A 0.000,B 0.000,C 90.000,E1 78.409} C_DIS
LIN {X 0.111,Y -578.453,Z 791.228,A 0.000,B 0.000,C 90.000,E1 77.061} C_DIS
LIN {X 0.207,Y -578.329,Z 791.221,A 0.000,B 0.000,C 90.000,E1 75.700} C_DIS
LIN {X 0.322,Y -577.946,Z 791.210,A 0.000,B 0.000,C 90.000,E1 73.795} C_DIS
LIN {X -0.153,Y -577.656,Z 791.203,A 0.000,B 0.000,C 90.000,E1 72.489} C_DIS
LIN {X -0.113,Y -577.360,Z 791.197,A 0.000,B 0.000,C 90.000,E1 71.402} C_DIS
LIN {X 0.132,Y -576.685,Z 791.188,A 0.000,B 0.000,C 90.000,E1 69.752} C_DIS
LIN {X -0.171,Y -575.925,Z 791.179,A 0.000,B 0.000,C 90.000,E1 68.156} C_DIS
LIN {X 0.254,Y -574.992,Z 791.170,A 0.000,B 0.000,C 90.000,E1 66.485} C_DIS
LIN {X 0.359,Y -573.871,Z 791.161,A 0.000,B 0.000,C 90.000,E1 64.845} C_DIS
LIN {X 0.243,Y -572.957,Z 791.154,A 0.000,B 0.000,C 90.000,E1 63.768} C_DIS
LIN {X 0.106,Y -571.943,Z 791.148,A 0.000,B 0.000,C 90.000,E1 62.692} C_DIS
LIN {X -0.124,Y -571.026,Z 791.144,A 0.000,B 0.000,C 90.000,E1 61.897} C_DIS
LIN {X -0.202,Y -569.171,Z 791.136,A 0.000,B 0.000,C 90.000,E1 60.539} C_DIS
LIN {X 0.143,Y -567.486,Z 791.130,A 0.000,B 0.000,C 90.000,E1 59.410} C_DIS
LIN {X -0.125,Y -566.069,Z 791.126,A 0.000,B 0.000,C 90.000,E1 58.614} C_DIS
LIN {X -0.110,Y -564.498,Z 791.121,A 0.000,B 0.000,C 90.000,E1 57.788} C_DIS
LIN {X -0.107,Y -562.709,Z 791.116,A 0.000,B 0.000,C 90.000,E1 56.962} C_DIS
LIN {X -0.337,Y -560.016,Z 791.110,A 0.000,B 0.000,C 90.000,E1 55.881} C_DIS
LIN {X -0.063,Y -557.767,Z 791.106,A 0.000,B 0.000,C 90.000,E1 55.022} C_DIS
LIN {X -0.132,Y -555.295,Z 791.101,A 0.000,B 0.000,C 90.000,E1 54.196} C_DIS
LIN {X 0.022,Y -553.603,Z 791.098,A 0.000,B 0.000,C 90.000,E1 53.623} C_DIS
LIN {X 0.230,Y -550.584,Z 791.093,A 0.000,B 0.000,C 90.000,E1 52.763} C_DIS
LIN {X -0.028,Y -547.320,Z 791.089,A 0.000,B 0.000,C 90.000,E1 51.949} C_DIS
LIN {X 0.109,Y -543.719,Z 791.084,A 0.000,B 0.000,C 90.000,E1 51.090} C_DIS
LIN {X -0.015,Y -541.801,Z 791.082,A 0.000,B 0.000,C 90.000,E1 50.678} C_DIS
LIN {X -0.206,Y -538.200,Z 791.078,A 0.000,B 0.000,C 90.000,E1 49.989} C_DIS
LIN {X 0.158,Y -535.120,Z 791.074,A 0.000,B 0.000,C 90.000,E1 49.380} C_DIS
LIN {X -0.255,Y -531.762,Z 791.071,A 0.000,B 0.000,C 90.000,E1 48.852} C_DIS
LIN {X 0.059,Y -527.935,Z 791.068,A 0.000,B 0.000,C 90.000,E1 48.243} C_DIS
LIN {X -0.049,Y -523.724,Z 791.065,A 0.000,B 0.000,C 90.000,E1 47.676} C_DIS
LIN {X 0.201,Y -519.042,Z 791.062,A 0.000,B 0.000,C 90.000,E1 47.067} C_DIS
LIN {X 0.045,Y -513.943,Z 791.058,A 0.000,B 0.000,C 90.000,E1 46.500} C_DIS
LIN {X 0.184,Y -509.932,Z 791.056,A 0.000,B 0.000,C 90.000,E1 46.053} C_DIS
LIN {X 0.128,Y -505.822,Z 791.054,A 0.000,B 0.000,C 90.000,E1 45.648} C_DIS
LIN {X 0.004,Y -499.065,Z 791.050,A 0.000,B 0.000,C 90.000,E1 45.040} C_DIS
LIN {X -0.153,Y -494.728,Z 791.048,A 0.000,B 0.000,C 90.000,E1 44.676} C_DIS
LIN {X 0.300,Y -487.313,Z 791.045,A 0.000,B 0.000,C 90.000,E1 44.028} C_DIS
LIN {X 0.084,Y -479.473,Z 791.042,A 0.000,B 0.000,C 90.000,E1 43.461} C_DIS
LIN {X -0.310,Y -466.632,Z 791.037,A 0.000,B 0.000,C 90.000,E1 42.609} C_DIS
LIN {X 0.042,Y -450.548,Z 791.030,A 0.000,B 0.000,C 90.000,E1 41.472} C_DIS
LIN {X 0.002,Y -420.402,Z 791.018,A 0.000,B 0.000,C 90.000,E1 39.277} C_DIS
LIN {X 0.065,Y -409.746,Z 791.013,A 0.000,B 0.000,C 90.000,E1 38.382} C_DIS
LIN {X -0.124,Y -404.498,Z 791.010,A 0.000,B 0.000,C 90.000,E1 37.890} C_DIS
LIN {X -0.155,Y -404.485,Z 791.010,A 0.000,B 0.000,C 90.000,E1 37.890} C_DIS
LIN {X -0.072,Y -395.903,Z 790.985,A 0.000,B 0.000,C 90.000,E1 33.293} C_DIS
LIN {X 0.137,Y -395.719,Z 790.984,A 0.000,B 0.000,C 90.000,E1 33.086} C_DIS
LIN {X -0.016,Y -396.462,Z 790.969,A 0.000,B 0.000,C 90.000,E1 30.463} C_DIS
LIN {X 0.008,Y -397.814,Z 790.954,A 0.000,B 0.000,C 90.000,E1 27.641} C_DIS
LIN {X 0.186,Y -399.261,Z 790.940,A 0.000,B 0.000,C 90.000,E1 25.155} C_DIS
LIN {X 0.077,Y -400.947,Z 790.926,A 0.000,B 0.000,C 90.000,E1 22.717} C_DIS
LIN {X 0.049,Y -403.672,Z 790.909,A 0.000,B 0.000,C 90.000,E1 19.577} C_DIS
LIN {X 0.208,Y -407.770,Z 790.890,A 0.000,B 0.000,C 90.000,E1 16.079} C_DIS
LIN {X -0.038,Y -412.362,Z 790.872,A 0.000,B 0.000,C 90.000,E1 13.008} C_DIS
LIN {X 0.007,Y -416.451,Z 790.859,A 0.000,B 0.000,C 90.000,E1 10.602} C_DIS
LIN {X -0.062,Y -420.014,Z 790.848,A 0.000,B 0.000,C 90.000,E1 8.568} C_DIS
LIN {X -0.115,Y -423.629,Z 790.836,A 0.000,B 0.000,C 90.000,E1 6.543} C_DIS
LIN {X -0.124,Y -427.919,Z 790.823,A 0.000,B 0.000,C 90.000,E1 4.188} C_DIS
LIN {X -0.104,Y -431.715,Z 790.812,A 0.000,B 0.000,C 90.000,E1 2.178} C_DIS
LIN {X 0.165,Y -436.496,Z 790.799,A 0.000,B 0.000,C 90.000,E1 359.771} C_DIS
LIN {X 0.168,Y -442.220,Z 790.784,A 0.000,B 0.000,C 90.000,E1 357.135} C_DIS
LIN {X -0.192,Y -447.613,Z 790.772,A 0.000,B 0.000,C 90.000,E1 354.894} C_DIS
LIN {X -0.062,Y -452.288,Z 790.761,A 0.000,B 0.000,C 90.000,E1 352.932} C_DIS
LIN {X 0.173,Y -456.891,Z 790.750,A 0.000,B 0.000,C 90.000,E1 350.971} C_DIS
LIN {X -0.012,Y -462.333,Z 790.738,A 0.000,B 0.000,C 90.000,E1 348.757} C_DIS
LIN {X 0.026,Y -464.333,Z 790.734,A 0.000,B 0.000,C 90.000,E1 348.117} C_DIS
LIN {X 0.001,Y -466.237,Z 790.731,A 0.000,B 0.000,C 90.000,E1 347.645} C_DIS
LIN {X -0.196,Y -467.825,Z 790.730,A 0.000,B 0.000,C 90.000,E1 347.353} C_DIS
LIN {X -0.082,Y -471.301,Z 790.727,A 0.000,B 0.000,C 90.000,E1 346.825} C_DIS
LIN {X -0.023,Y -475.459,Z 790.724,A 0.000,B 0.000,C 90.000,E1 346.353} C_DIS
LIN {X -0.017,Y -481.892,Z 790.721,A 0.000,B 0.000,C 90.000,E1 345.755} C_DIS
LIN {X -0.051,Y -496.085,Z 790.715,A 0.000,B 0.000,C 90.000,E1 344.700} C_DIS
LIN {X -0.208,Y -510.373,Z 790.710,A 0.000,B 0.000,C 90.000,E1 343.740} C_DIS
LIN {X -0.162,Y -529.360,Z 790.703,A 0.000,B 0.000,C 90.000,E1 342.472} C_DIS
LIN {X -0.100,Y -537.014,Z 790.700,A 0.000,B 0.000,C 90.000,E1 341.945} C_DIS
LIN {X 0.094,Y -547.597,Z 790.695,A 0.000,B 0.000,C 90.000,E1 341.167} C_DIS
LIN {X -0.114,Y -552.053,Z 790.694,A 0.000,B 0.000,C 90.000,E1 340.859} C_DIS
LIN {X 0.068,Y -556.381,Z 790.692,A 0.000,B 0.000,C 90.000,E1 340.496} C_DIS
LIN {X 0.180,Y -561.809,Z 790.689,A 0.000,B 0.000,C 90.000,E1 340.007} C_DIS
LIN {X 0.017,Y -567.010,Z 790.686,A 0.000,B 0.000,C 90.000,E1 339.518} C_DIS
LIN {X 0.143,Y -571.943,Z 790.683,A 0.000,B 0.000,C 90.000,E1 338.975} C_DIS
LIN {X 0.271,Y -577.623,Z 790.680,A 0.000,B 0.000,C 90.000,E1 338.284} C_DIS
LIN {X 0.140,Y -583.965,Z 790.675,A 0.000,B 0.000,C 90.000,E1 337.486} C_DIS
LIN {X -0.182,Y -588.847,Z 790.671,A 0.000,B 0.000,C 90.000,E1 336.847} C_DIS
LIN {X -0.258,Y -595.332,Z 790.666,A 0.000,B 0.000,C 90.000,E1 335.921} C_DIS
LIN {X -0.050,Y -602.319,Z 790.660,A 0.000,B 0.000,C 90.000,E1 334.845} C_DIS
LIN {X 0.258,Y -608.855,Z 790.654,A 0.000,B 0.000,C 90.000,E1 333.768} C_DIS
LIN {X 0.108,Y -614.971,Z 790.649,A 0.000,B 0.000,C 90.000,E1 332.743} C_DIS
LIN {X 0.044,Y -619.365,Z 790.644,A 0.000,B 0.000,C 90.000,E1 331.975} C_DIS
LIN {X 0.322,Y -625.057,Z 790.639,A 0.000,B 0.000,C 90.000,E1 330.923} C_DIS
LIN {X 0.139,Y -630.485,Z 790.633,A 0.000,B 0.000,C 90.000,E1 329.921} C_DIS
LIN {X -0.329,Y -634.234,Z 790.629,A 0.000,B 0.000,C 90.000,E1 329.203} C_DIS
LIN {X 0.104,Y -637.878,Z 790.625,A 0.000,B 0.000,C 90.000,E1 328.408} C_DIS
LIN {X 0.073,Y -642.418,Z 790.619,A 0.000,B 0.000,C 90.000,E1 327.406} C_DIS
LIN {X 0.391,Y -645.696,Z 790.615,A 0.000,B 0.000,C 90.000,E1 326.628} C_DIS
LIN {X 0.349,Y -650.683,Z 790.608,A 0.000,B 0.000,C 90.000,E1 325.388} C_DIS
LIN {X -0.143,Y -653.490,Z 790.604,A 0.000,B 0.000,C 90.000,E1 324.689} C_DIS
LIN {X 0.313,Y -657.900,Z 790.597,A 0.000,B 0.000,C 90.000,E1 323.417} C_DIS
LIN {X 0.316,Y -661.909,Z 790.590,A 0.000,B 0.000,C 90.000,E1 322.190} C_DIS
LIN {X 0.358,Y -666.303,Z 790.582,A 0.000,B 0.000,C 90.000,E1 320.723} C_DIS
LIN {X -0.031,Y -670.286,Z 790.574,A 0.000,B 0.000,C 90.000,E1 319.299} C_DIS
LIN {X 0.077,Y -673.334,Z 790.567,A 0.000,B 0.000,C 90.000,E1 318.081} C_DIS
LIN {X -0.339,Y -674.558,Z 790.565,A 0.000,B 0.000,C 90.000,E1 317.634} C_DIS
LIN {X 0.286,Y -677.127,Z 790.558,A 0.000,B 0.000,C 90.000,E1 316.377} C_DIS
LIN {X 0.031,Y -679.721,Z 790.550,A 0.000,B 0.000,C 90.000,E1 314.960} C_DIS
LIN {X -0.319,Y -680.993,Z 790.546,A 0.000,B 0.000,C 90.000,E1 314.271} C_DIS
LIN {X -0.030,Y -683.199,Z 790.538,A 0.000,B 0.000,C 90.000,E1 312.813} C_DIS
LIN {X 0.276,Y -684.892,Z 790.531,A 0.000,B 0.000,C 90.000,E1 311.595} C_DIS
LIN {X 0.039,Y -686.104,Z 790.526,A 0.000,B 0.000,C 90.000,E1 310.663} C_DIS
LIN {X -0.050,Y -687.440,Z 790.519,A 0.000,B 0.000,C 90.000,E1 309.483} C_DIS
LIN {X -0.116,Y -688.655,Z 790.513,A 0.000,B 0.000,C 90.000,E1 308.302} C_DIS
LIN {X 0.012,Y -690.039,Z 790.505,A 0.000,B 0.000,C 90.000,E1 306.870} C_DIS
LIN {X 0.166,Y -691.284,Z 790.497,A 0.000,B 0.000,C 90.000,E1 305.438} C_DIS
LIN {X -0.096,Y -692.164,Z 790.490,A 0.000,B 0.000,C 90.000,E1 304.278} C_DIS
LIN {X -0.080,Y -693.408,Z 790.481,A 0.000,B 0.000,C 90.000,E1 302.625} C_DIS
LIN {X 0.184,Y -694.894,Z 790.471,A 0.000,B 0.000,C 90.000,E1 300.718} C_DIS
LIN {X 0.219,Y -695.612,Z 790.464,A 0.000,B 0.000,C 90.000,E1 299.539} C_DIS
LIN {X 0.168,Y -696.487,Z 790.455,A 0.000,B 0.000,C 90.000,E1 297.897} C_DIS
LIN {X -0.199,Y -697.414,Z 790.446,A 0.000,B 0.000,C 90.000,E1 296.283} C_DIS
LIN {X 0.145,Y -698.331,Z 790.438,A 0.000,B 0.000,C 90.000,E1 294.847} C_DIS
LIN {X 0.014,Y -698.497,Z 790.434,A 0.000,B 0.000,C 90.000,E1 294.155} C_DIS
LIN {X -0.098,Y -697.696,Z 790.432,A 0.000,B 0.000,C 90.000,E1 293.695} C_DIS
LIN {X -0.117,Y -697.114,Z 790.430,A 0.000,B 0.000,C 90.000,E1 293.462} C_DIS
LIN {X 0.141,Y -695.741,Z 790.429,A 0.000,B 0.000,C 90.000,E1 293.206} C_DIS
LIN {X 0.393,Y -694.116,Z 790.428,A 0.000,B 0.000,C 90.000,E1 292.950} C_DIS
LIN {X -0.269,Y -692.190,Z 790.426,A 0.000,B 0.000,C 90.000,E1 292.770} C_DIS
LIN {X -0.148,Y -690.640,Z 790.426,A 0.000,B 0.000,C 90.000,E1 292.642} C_DIS
LIN {X 0.225,Y -684.970,Z 790.424,A 0.000,B 0.000,C 90.000,E1 292.333} C_DIS
LIN {X -0.042,Y -683.294,Z 790.424,A 0.000,B 0.000,C 90.000,E1 292.280} C_DIS
LIN {X -0.048,Y -681.226,Z 790.423,A 0.000,B 0.000,C 90.000,E1 292.206} C_DIS
LIN {X 0.038,Y -675.111,Z 790.422,A 0.000,B 0.000,C 90.000,E1 292.025} C_DIS
LIN {X 0.073,Y -673.050,Z 790.422,A 0.000,B 0.000,C 90.000,E1 291.972} C_DIS
LIN {X 0.158,Y -649.930,Z 790.420,A 0.000,B 0.000,C 90.000,E1 291.589} C_DIS
LIN {X -0.030,Y -632.910,Z 790.418,A 0.000,B 0.000,C 90.000,E1 291.280} C_DIS
LIN {X 0.287,Y -612.289,Z 790.416,A 0.000,B 0.000,C 90.000,E1 290.791} C_DIS
LIN {X -0.075,Y -595.348,Z 790.413,A 0.000,B 0.000,C 90.000,E1 290.375} C_DIS
LIN {X -0.186,Y -578.445,Z 790.410,A 0.000,B 0.000,C 90.000,E1 289.866} C_DIS
LIN {X -0.063,Y -572.180,Z 790.409,A 0.000,B 0.000,C 90.000,E1 289.631} C_DIS
LIN {X -0.089,Y -564.921,Z 790.407,A 0.000,B 0.000,C 90.000,E1 289.322} C_DIS
LIN {X -0.279,Y -563.462,Z 790.407,A 0.000,B 0.000,C 90.000,E1 289.268} C_DIS
LIN {X 0.318,Y -560.114,Z 790.406,A 0.000,B 0.000,C 90.000,E1 288.960} C_DIS
LIN {X -0.216,Y -559.538,Z 790.405,A 0.000,B 0.000,C 90.000,E1 288.960} C_DIS
LIN {X -0.156,Y -557.658,Z 790.404,A 0.000,B 0.000,C 90.000,E1 288.671} C_DIS
LIN {X 0.024,Y -555.986,Z 790.401,A 0.000,B 0.000,C 90.000,E1 288.236} C_DIS
LIN {X -0.171,Y -555.252,Z 790.400,A 0.000,B 0.000,C 90.000,E1 287.928} C_DIS
LIN {X 0.056,Y -554.392,Z 790.396,A 0.000,B 0.000,C 90.000,E1 287.347} C_DIS
LIN {X 0.056,Y -552.754,Z 790.376,A 0.000,B 0.000,C 90.000,E1 283.716} C_DIS
LIN {X 0.243,Y -552.285,Z 790.369,A 0.000,B 0.000,C 90.000,E1 282.299} C_DIS
LIN {X 0.103,Y -551.581,Z 790.356,A 0.000,B 0.000,C 90.000,E1 280.074} C_DIS
LIN {X -0.224,Y -550.988,Z 790.342,A 0.000,B 0.000,C 90.000,E1 277.587} C_DIS
LIN {X 0.133,Y -550.543,Z 790.336,A 0.000,B 0.000,C 90.000,E1 276.429} C_DIS
LIN {X -0.085,Y -549.842,Z 790.328,A 0.000,B 0.000,C 90.000,E1 275.049} C_DIS
LIN {X 0.186,Y -549.164,Z 790.322,A 0.000,B 0.000,C 90.000,E1 273.898} C_DIS
LIN {X 0.069,Y -547.713,Z 790.309,A 0.000,B 0.000,C 90.000,E1 271.661} C_DIS
LIN {X -0.247,Y -546.766,Z 790.302,A 0.000,B 0.000,C 90.000,E1 270.286} C_DIS
LIN {X -0.031,Y -545.829,Z 790.294,A 0.000,B 0.000,C 90.000,E1 268.854} C_DIS
LIN {X 0.246,Y -544.470,Z 790.283,A 0.000,B 0.000,C 90.000,E1 266.849} C_DIS
LIN {X 0.010,Y -543.281,Z 790.272,A 0.000,B 0.000,C 90.000,E1 264.894} C_DIS
LIN {X 0.200,Y -542.341,Z 790.264,A 0.000,B 0.000,C 90.000,E1 263.457} C_DIS
LIN {X -0.111,Y -541.424,Z 790.258,A 0.000,B 0.000,C 90.000,E1 262.356} C_DIS
LIN {X 0.239,Y -539.732,Z 790.246,A 0.000,B 0.000,C 90.000,E1 260.330} C_DIS
LIN {X -0.006,Y -538.729,Z 790.240,A 0.000,B 0.000,C 90.000,E1 259.218} C_DIS
LIN {X -0.127,Y -537.071,Z 790.231,A 0.000,B 0.000,C 90.000,E1 257.521} C_DIS
LIN {X 0.170,Y -535.681,Z 790.223,A 0.000,B 0.000,C 90.000,E1 256.061} C_DIS
LIN {X 0.221,Y -533.779,Z 790.213,A 0.000,B 0.000,C 90.000,E1 254.338} C_DIS
LIN {X -0.024,Y -532.773,Z 790.208,A 0.000,B 0.000,C 90.000,E1 253.504} C_DIS
LIN {X 0.094,Y -531.131,Z 790.200,A 0.000,B 0.000,C 90.000,E1 252.054} C_DIS
LIN {X 0.001,Y -529.774,Z 790.194,A 0.000,B 0.000,C 90.000,E1 250.913} C_DIS
LIN {X 0.241,Y -527.780,Z 790.186,A 0.000,B 0.000,C 90.000,E1 249.444} C_DIS
LIN {X -0.043,Y -525.723,Z 790.178,A 0.000,B 0.000,C 90.000,E1 248.028} C_DIS
LIN {X -0.053,Y -523.963,Z 790.172,A 0.000,B 0.000,C 90.000,E1 246.869} C_DIS
LIN {X 0.000,Y -521.758,Z 790.163,A 0.000,B 0.000,C 90.000,E1 245.409} C_DIS
LIN {X 0.023,Y -519.394,Z 790.155,A 0.000,B 0.000,C 90.000,E1 243.948} C_DIS
LIN {X -0.129,Y -517.457,Z 790.149,A 0.000,B 0.000,C 90.000,E1 242.794} C_DIS
LIN {X 0.024,Y -515.936,Z 790.144,A 0.000,B 0.000,C 90.000,E1 241.897} C_DIS
LIN {X 0.159,Y -513.183,Z 790.136,A 0.000,B 0.000,C 90.000,E1 240.411} C_DIS
LIN {X 0.043,Y -510.440,Z 790.128,A 0.000,B 0.000,C 90.000,E1 238.948} C_DIS
LIN {X -0.184,Y -508.019,Z 790.121,A 0.000,B 0.000,C 90.000,E1 237.788} C_DIS
LIN {X -0.230,Y -504.292,Z 790.111,A 0.000,B 0.000,C 90.000,E1 236.008} C_DIS
LIN {X 0.153,Y -501.557,Z 790.104,A 0.000,B 0.000,C 90.000,E1 234.769} C_DIS
LIN {X -0.201,Y -499.394,Z 790.099,A 0.000,B 0.000,C 90.000,E1 233.909} C_DIS
LIN {X -0.138,Y -495.629,Z 790.091,A 0.000,B 0.000,C 90.000,E1 232.396} C_DIS
LIN {X -0.141,Y -490.358,Z 790.079,A 0.000,B 0.000,C 90.000,E1 230.275} C_DIS
LIN {X -0.059,Y -484.086,Z 790.064,A 0.000,B 0.000,C 90.000,E1 227.514} C_DIS
LIN {X 0.091,Y -480.123,Z 790.054,A 0.000,B 0.000,C 90.000,E1 225.648} C_DIS
LIN {X 0.019,Y -476.706,Z 790.045,A 0.000,B 0.000,C 90.000,E1 224.109} C_DIS
LIN {X 0.222,Y -473.288,Z 790.036,A 0.000,B 0.000,C 90.000,E1 222.528} C_DIS
LIN {X 0.008,Y -467.943,Z 790.023,A 0.000,B 0.000,C 90.000,E1 220.048} C_DIS
LIN {X -0.164,Y -463.966,Z 790.012,A 0.000,B 0.000,C 90.000,E1 218.177} C_DIS
LIN {X -0.104,Y -460.713,Z 790.003,A 0.000,B 0.000,C 90.000,E1 216.583} C_DIS
LIN {X 0.198,Y -455.343,Z 789.989,A 0.000,B 0.000,C 90.000,E1 213.992} C_DIS
LIN {X -0.063,Y -452.150,Z 789.980,A 0.000,B 0.000,C 90.000,E1 212.418} C_DIS
LIN {X 0.076,Y -448.328,Z 789.969,A 0.000,B 0.000,C 90.000,E1 210.463} C_DIS
LIN {X -0.112,Y -444.552,Z 789.958,A 0.000,B 0.000,C 90.000,E1 208.537} C_DIS
LIN {X -0.022,Y -440.840,Z 789.948,A 0.000,B 0.000,C 90.000,E1 206.565} C_DIS
LIN {X 0.155,Y -437.691,Z 789.938,A 0.000,B 0.000,C 90.000,E1 204.899} C_DIS
